KUKA KRL program: MyProgram_286().src

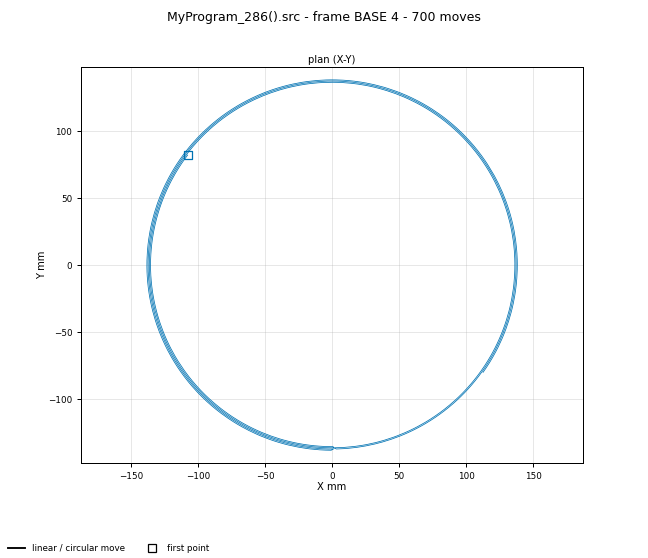
[picture p0: tool path of MyProgram_286().src in frame BASE 4, 700 of 700 moves have a stored position in this frame; points joined in program order, loops and branches not executed]
&ACCESS RVP
&REL 1
&PARAM TEMPLATE = C:\KRC\Roboter\Template\vorgabe
&PARAM EDITMASK = *
DEF MyProgram_286()
; ---- Setting reference (Base) ----
$BASE = BASE_DATA[4]

; --------------------------
; ---- Setting tool (TCP) ----
$TOOL = TOOL_DATA[3]
; --------------------------

$VEL.CP = VEL_APROX_PRINT
Startdeposition()
$VEL.CP = VEL_PRINT
LIN {X -107.8161,Y 82.1036,Z 175,A 144.1909,B 7.7185,C 0.1513,E1 7.5924,E2 307.6378} C_DIS
LIN {X -110.1334,Y 78.9678,Z 175,A 146.0967,B 7.7185,C 0.1516,E1 7.5892,E2 305.7022} C_DIS
LIN {X -112.383,Y 75.7323,Z 175,A 147.6376,B 7.7183,C 0.1573,E1 7.5868,E2 304.1782} C_DIS
LIN {X -114.7272,Y 72.1316,Z 175,A 149.9305,B 7.7183,C 0.1551,E1 7.5833,E2 301.8286} C_DIS
LIN {X -117.0253,Y 68.3406,Z 175,A 151.2224,B 7.7181,C 0.1679,E1 7.5816,E2 300.61} C_DIS
LIN {X -120.0251,Y 62.9181,Z 175,A 153.9854,B 7.718,C 0.1726,E1 7.5779,E2 297.8322} C_DIS
LIN {X -121.646,Y 59.7246,Z 175,A 155.5473,B 7.718,C 0.1759,E1 7.5759,E2 296.2659} C_DIS
LIN {X -123.0692,Y 56.7336,Z 175,A 156.9832,B 7.7179,C 0.179,E1 7.5742,E2 294.8271} C_DIS
LIN {X -124.7084,Y 53.0394,Z 175,A 158.6778,B 7.7177,C 0.1838,E1 7.5723,E2 293.136} C_DIS
LIN {X -126.0542,Y 49.7548,Z 175,A 160.6289,B 7.7177,C 0.1817,E1 7.5703,E2 291.1309} C_DIS
LIN {X -127.3827,Y 46.2436,Z 175,A 162.2434,B 7.7177,C 0.1856,E1 7.5687,E2 289.5146} C_DIS
LIN {X -128.6415,Y 42.6164,Z 175,A 163.4802,B 7.7175,C 0.1953,E1 7.5677,E2 288.327} C_DIS
LIN {X -129.7186,Y 39.2178,Z 175,A 165.0342,B 7.7174,C 0.1989,E1 7.5664,E2 286.7687} C_DIS
LIN {X -130.9414,Y 34.9158,Z 175,A 167.0103,B 7.7173,C 0.203,E1 7.5649,E2 284.7839} C_DIS
LIN {X -131.9367,Y 30.9533,Z 175,A 168.8678,B 7.7172,C 0.2061,E1 7.5637,E2 282.9121} C_DIS
LIN {X -132.7918,Y 27.039,Z 175,A 170.4341,B 7.717,C 0.2126,E1 7.5628,E2 281.363} C_DIS
LIN {X -133.4946,Y 23.33,Z 175,A 172.024,B 7.7169,C 0.2172,E1 7.562,E2 279.7755} C_DIS
LIN {X -134.0907,Y 19.6137,Z 175,A 173.7622,B 7.7169,C 0.2198,E1 7.5613,E2 278.0206} C_DIS
LIN {X -134.5829,Y 15.8836,Z 175,A 175.3324,B 7.7167,C 0.2246,E1 7.5607,E2 276.4544} C_DIS
LIN {X -135.012,Y 11.691,Z 175,A 177.1354,B 7.7165,C 0.2295,E1 7.5602,E2 274.6504} C_DIS
LIN {X -135.2718,Y 8.1499,Z 175,A 178.6452,B 7.7164,C 0.2337,E1 7.56,E2 273.1409} C_DIS
LIN {X -135.4563,Y 4.0677,Z 175,A -179.5523,B 7.7163,C 0.2376,E1 7.5598,E2 271.3307} C_DIS
LIN {X -135.5184,Y 0.2685,Z 175,A -177.968,B 7.7161,C 0.2426,E1 7.5598,E2 269.7506} C_DIS
LIN {X -135.4713,Y -3.5254,Z 175,A -176.2406,B 7.7161,C 0.2455,E1 7.5598,E2 268.0093} C_DIS
LIN {X -135.3015,Y -7.6668,Z 175,A -174.4134,B 7.7159,C 0.2496,E1 7.5601,E2 266.1745} C_DIS
LIN {X -135.0006,Y -11.8252,Z 175,A -172.6182,B 7.7158,C 0.2542,E1 7.5605,E2 264.3766} C_DIS
LIN {X -134.5616,Y -16.0623,Z 175,A -170.8656,B 7.7156,C 0.26,E1 7.561,E2 262.6314} C_DIS
LIN {X -133.9782,Y -20.3659,Z 175,A -168.9506,B 7.7154,C 0.2641,E1 7.5618,E2 260.7082} C_DIS
LIN {X -133.3593,Y -24.0861,Z 175,A -167.4144,B 7.7152,C 0.2694,E1 7.5625,E2 259.1805} C_DIS
LIN {X -132.7048,Y -27.4669,Z 175,A -165.9397,B 7.7152,C 0.2733,E1 7.5633,E2 257.7045} C_DIS
LIN {X -131.904,Y -31.0896,Z 175,A -163.8821,B 7.7152,C 0.2709,E1 7.5647,E2 255.5872} C_DIS
LIN {X -130.9675,Y -34.818,Z 175,A -162.2439,B 7.715,C 0.2752,E1 7.5658,E2 253.9485} C_DIS
LIN {X -129.9083,Y -38.5844,Z 175,A -160.7008,B 7.7148,C 0.2813,E1 7.567,E2 252.4205} C_DIS
LIN {X -128.4088,Y -43.3151,Z 175,A -158.7744,B 7.7145,C 0.2894,E1 7.5687,E2 250.517} C_DIS
LIN {X -127.31,Y -46.4452,Z 175,A -157.4935,B 7.7143,C 0.2948,E1 7.5699,E2 249.2522} C_DIS
LIN {X -126.257,Y -49.2333,Z 175,A -156.1015,B 7.7143,C 0.2963,E1 7.5713,E2 247.8446} C_DIS
LIN {X -124.9108,Y -52.5561,Z 175,A -154.5532,B 7.7141,C 0.2999,E1 7.573,E2 246.2932} C_DIS
LIN {X -123.4445,Y -55.9159,Z 175,A -152.6719,B 7.7141,C 0.2993,E1 7.5752,E2 244.3714} C_DIS
LIN {X -121.9662,Y -59.0717,Z 175,A -151.5247,B 7.7138,C 0.3076,E1 7.5765,E2 243.2659} C_DIS
LIN {X -120.4316,Y -62.1407,Z 175,A -150.0468,B 7.7137,C 0.3109,E1 7.5784,E2 241.7855} C_DIS
LIN {X -117.2772,Y -67.9066,Z 175,A -147.4697,B 7.7133,C 0.3207,E1 7.5818,E2 239.2352} C_DIS
LIN {X -114.8122,Y -71.997,Z 175,A -145.0301,B 7.7133,C 0.3196,E1 7.5854,E2 236.744} C_DIS
LIN {X -110.3112,Y -78.7191,Z 175,A -140.919,B 7.7134,C 0.3176,E1 7.5921,E2 232.5474} C_DIS
LIN {X -106.8941,Y -83.3008,Z 175,A -139.1429,B 7.7128,C 0.3322,E1 7.595,E2 230.8533} C_DIS
LIN {X -104.2988,Y -86.5276,Z 175,A -137.3671,B 7.7127,C 0.3357,E1 7.5981,E2 229.075} C_DIS
LIN {X -101.2925,Y -90.0288,Z 175,A -135.503,B 7.7124,C 0.341,E1 7.6015,E2 227.2226} C_DIS
LIN {X -98.2121,Y -93.3795,Z 175,A -133.4036,B 7.7124,C 0.3424,E1 7.6056,E2 225.1017} C_DIS
LIN {X -95.0625,Y -96.5837,Z 175,A -131.5003,B 7.7122,C 0.3461,E1 7.6093,E2 223.1985} C_DIS
LIN {X -91.4043,Y -100.0534,Z 175,A -129.4346,B 7.712,C 0.3511,E1 7.6135,E2 221.1417} C_DIS
LIN {X -88.3999,Y -102.7166,Z 175,A -127.6314,B 7.712,C 0.3526,E1 7.6173,E2 219.3255} C_DIS
LIN {X -84.3117,Y -106.098,Z 175,A -125.4213,B 7.7117,C 0.357,E1 7.6221,E2 217.1201} C_DIS
LIN {X -81.0086,Y -108.6409,Z 175,A -123.1556,B 7.7119,C 0.3522,E1 7.6273,E2 214.7909} C_DIS
LIN {X -77.435,Y -111.2163,Z 175,A -121.831,B 7.7114,C 0.3634,E1 7.6302,E2 213.5347} C_DIS
LIN {X -74.2923,Y -113.3401,Z 175,A -120.0625,B 7.7114,C 0.3633,E1 7.6343,E2 211.7454} C_DIS
LIN {X -70.4646,Y -115.759,Z 175,A -118.111,B 7.7114,C 0.3654,E1 7.639,E2 209.7894} C_DIS
LIN {X -66.6771,Y -117.981,Z 175,A -116.2393,B 7.7112,C 0.3677,E1 7.6435,E2 207.9158} C_DIS
LIN {X -62.6258,Y -120.1786,Z 175,A -114.4226,B 7.711,C 0.3722,E1 7.648,E2 206.1158} C_DIS
LIN {X -59.8693,Y -121.5745,Z 175,A -113.0442,B 7.711,C 0.3726,E1 7.6514,E2 204.7282} C_DIS
LIN {X -56.0366,Y -123.3904,Z 175,A -111.0915,B 7.711,C 0.372,E1 7.6564,E2 202.7552} C_DIS
LIN {X -52.1981,Y -125.0603,Z 175,A -109.5877,B 7.7107,C 0.3781,E1 7.6602,E2 201.285} C_DIS
LIN {X -48.4755,Y -126.5515,Z 175,A -107.7935,B 7.7107,C 0.3781,E1 7.6649,E2 199.4781} C_DIS
LIN {X -45.5877,Y -127.6192,Z 175,A -106.472,B 7.7107,C 0.3789,E1 7.6684,E2 198.1538} C_DIS
LIN {X -39.2294,Y -129.7151,Z 175,A -103.6522,B 7.7106,C 0.3813,E1 7.6759,E2 195.3351} C_DIS
LIN {X -36.0972,Y -130.6213,Z 175,A -102.2133,B 7.7106,C 0.3813,E1 7.6798,E2 193.8882} C_DIS
LIN {X -32.0637,Y -131.6692,Z 175,A -100.4417,B 7.7106,C 0.3821,E1 7.6846,E2 192.115} C_DIS
LIN {X -28.348,Y -132.5188,Z 175,A -98.8307,B 7.7105,C 0.3829,E1 7.689,E2 190.5035} C_DIS
LIN {X -24.7465,Y -133.24,Z 175,A -97.2309,B 7.7105,C 0.3829,E1 7.6934,E2 188.8974} C_DIS
LIN {X -20.8968,Y -133.896,Z 175,A -95.5882,B 7.7105,C 0.3835,E1 7.6979,E2 187.2552} C_DIS
LIN {X -17.0911,Y -134.4352,Z 175,A -93.628,B 7.7107,C 0.3783,E1 7.7035,E2 185.2516} C_DIS
LIN {X -13.3209,Y -134.8611,Z 175,A -92.3436,B 7.7104,C 0.384,E1 7.7069,E2 184.0075} C_DIS
LIN {X -9.5355,Y -135.1814,Z 175,A -90.5074,B 7.7106,C 0.3803,E1 7.7121,E2 182.1413} C_DIS
LIN {X -6.1557,Y -135.3786,Z 175,A -89.3546,B 7.7104,C 0.385,E1 7.7152,E2 181.0235} C_DIS
LIN {X 0.789,Y -135.5147,Z 175,A -86.4061,B 7.7104,C 0.3846,E1 7.7235,E2 178.0722} C_DIS
LIN {X 0.789,Y -135.5147,Z 175,A -86.4061,B 7.7104,C 0.3846,E1 7.7235,E2 178.0722} C_DIS
Enddeposition()
LIN {X 1.0147,Y -136.4185,Z 175,A -86.3345,B 7.6595,C 0.3899,E1 7.673,E2 178.0513} C_DIS
Startdeposition()
$VEL.CP = VEL_PRINT
LIN {X -5.9801,Y -136.294,Z 175,A -89.7795,B 7.659,C 0.3988,E1 7.6632,E2 181.5627} C_DIS
LIN {X -12.1256,Y -135.885,Z 175,A -92.4451,B 7.659,C 0.3999,E1 7.6557,E2 184.2395} C_DIS
LIN {X -18.4218,Y -135.1756,Z 175,A -95.5048,B 7.6587,C 0.4059,E1 7.6471,E2 187.3506} C_DIS
LIN {X -22.0387,Y -134.632,Z 175,A -96.6557,B 7.659,C 0.399,E1 7.644,E2 188.4533} C_DIS
LIN {X -25.4217,Y -134.0338,Z 175,A -98.1167,B 7.659,C 0.3988,E1 7.64,E2 189.917} C_DIS
LIN {X -28.6784,Y -133.3748,Z 175,A -99.5243,B 7.659,C 0.3983,E1 7.6361,E2 191.3266} C_DIS
LIN {X -31.6236,Y -132.7078,Z 175,A -100.774,B 7.6591,C 0.3973,E1 7.6328,E2 192.5742} C_DIS
LIN {X -34.3363,Y -132.0338,Z 175,A -102.1182,B 7.6591,C 0.3994,E1 7.6291,E2 193.9403} C_DIS
LIN {X -38.6904,Y -130.8222,Z 175,A -103.9583,B 7.6591,C 0.3971,E1 7.6241,E2 195.7734} C_DIS
LIN {X -43.7485,Y -129.2199,Z 175,A -106.2507,B 7.6591,C 0.3964,E1 7.618,E2 198.0744} C_DIS
LIN {X -47.4516,Y -127.9053,Z 175,A -107.7892,B 7.6593,C 0.3932,E1 7.614,E2 199.599} C_DIS
LIN {X -50.3236,Y -126.8042,Z 175,A -109.1767,B 7.6593,C 0.3935,E1 7.6104,E2 200.9987} C_DIS
LIN {X -56.3141,Y -124.2593,Z 175,A -111.941,B 7.6594,C 0.3911,E1 7.6033,E2 203.7671} C_DIS
LIN {X -59.924,Y -122.5584,Z 175,A -113.5022,B 7.6596,C 0.3874,E1 7.5994,E2 205.3139} C_DIS
LIN {X -63.3045,Y -120.846,Z 175,A -115.1161,B 7.6597,C 0.3858,E1 7.5954,E2 206.9306} C_DIS
LIN {X -67.1452,Y -118.7577,Z 175,A -117.04,B 7.6597,C 0.3848,E1 7.5907,E2 208.8656} C_DIS
LIN {X -70.6813,Y -116.6873,Z 175,A -118.7791,B 7.6599,C 0.3827,E1 7.5865,E2 210.607} C_DIS
LIN {X -74.4795,Y -114.3005,Z 175,A -120.7118,B 7.6599,C 0.3807,E1 7.5819,E2 212.5456} C_DIS
LIN {X -78.1156,Y -111.8471,Z 175,A -122.6441,B 7.66,C 0.3792,E1 7.5774,E2 214.489} C_DIS
LIN {X -81.8071,Y -109.1766,Z 175,A -124.5295,B 7.6602,C 0.3757,E1 7.5732,E2 216.3707} C_DIS
LIN {X -85.157,Y -106.5838,Z 175,A -126.196,B 7.6604,C 0.371,E1 7.5696,E2 218.0227} C_DIS
LIN {X -88.185,Y -104.0924,Z 175,A -127.9779,B 7.6604,C 0.3701,E1 7.5657,E2 219.8212} C_DIS
LIN {X -91.4413,Y -101.2439,Z 175,A -129.638,B 7.6607,C 0.3645,E1 7.5623,E2 221.4612} C_DIS
LIN {X -94.0168,Y -98.857,Z 175,A -131.2904,B 7.6607,C 0.3643,E1 7.5589,E2 223.1355} C_DIS
LIN {X -97.1533,Y -95.7764,Z 175,A -133.1996,B 7.6609,C 0.3616,E1 7.5551,E2 225.0521} C_DIS
LIN {X -100.5029,Y -92.2547,Z 175,A -135.1908,B 7.6611,C 0.3567,E1 7.5513,E2 227.0363} C_DIS
LIN {X -103.7292,Y -88.6122,Z 175,A -137.3399,B 7.6612,C 0.3539,E1 7.5473,E2 229.1979} C_DIS
LIN {X -106.6969,Y -85.0149,Z 175,A -139.2989,B 7.6614,C 0.3497,E1 7.5439,E2 231.1562} C_DIS
LIN {X -110.2775,Y -80.3164,Z 175,A -141.8463,B 7.6616,C 0.345,E1 7.5396,E2 233.7109} C_DIS
LIN {X -112.9731,Y -76.4778,Z 175,A -143.9771,B 7.6617,C 0.3427,E1 7.5362,E2 235.8608} C_DIS
LIN {X -115.8349,Y -72.0696,Z 175,A -146.039,B 7.6621,C 0.3354,E1 7.5332,E2 237.9036} C_DIS
LIN {X -118.3923,Y -67.7871,Z 175,A -148.3088,B 7.6621,C 0.3328,E1 7.5299,E2 240.1939} C_DIS
LIN {X -120.522,Y -63.9216,Z 175,A -150.0817,B 7.6624,C 0.327,E1 7.5276,E2 241.9558} C_DIS
LIN {X -122.2542,Y -60.5406,Z 175,A -151.5848,B 7.6626,C 0.3217,E1 7.5257,E2 243.4465} C_DIS
LIN {X -123.5045,Y -57.9521,Z 175,A -152.9385,B 7.6626,C 0.3206,E1 7.5241,E2 244.8177} C_DIS
LIN {X -125.105,Y -54.4064,Z 175,A -154.5088,B 7.6629,C 0.3155,E1 7.5223,E2 246.3792} C_DIS
LIN {X -126.4585,Y -51.1811,Z 175,A -155.9996,B 7.663,C 0.3119,E1 7.5207,E2 247.8716} C_DIS
LIN {X -127.5287,Y -48.4571,Z 175,A -157.1831,B 7.6632,C 0.3081,E1 7.5195,E2 249.0488} C_DIS
LIN {X -128.4332,Y -46.0026,Z 175,A -158.7635,B 7.6631,C 0.3117,E1 7.518,E2 250.688} C_DIS
LIN {X -129.7192,Y -42.2465,Z 175,A -160.0232,B 7.6635,C 0.3016,E1 7.5169,E2 251.8963} C_DIS
LIN {X -132.1456,Y -33.8958,Z 175,A -163.9384,B 7.6637,C 0.2952,E1 7.514,E2 255.8416} C_DIS
LIN {X -133.2218,Y -29.3871,Z 175,A -165.8816,B 7.6639,C 0.2897,E1 7.5127,E2 257.7829} C_DIS
LIN {X -133.9192,Y -26.0215,Z 175,A -167.2777,B 7.6641,C 0.285,E1 7.512,E2 259.172} C_DIS
LIN {X -134.5511,Y -22.5233,Z 175,A -168.7249,B 7.6643,C 0.2802,E1 7.5113,E2 260.6125} C_DIS
LIN {X -135.0574,Y -19.2563,Z 175,A -170.2524,B 7.6643,C 0.2781,E1 7.5106,E2 262.156} C_DIS
LIN {X -135.5764,Y -15.19,Z 175,A -172.0277,B 7.6645,C 0.2739,E1 7.51,E2 263.9366} C_DIS
LIN {X -135.9437,Y -11.4309,Z 175,A -173.5577,B 7.6647,C 0.2686,E1 7.5097,E2 265.4583} C_DIS
LIN {X -136.2347,Y -7.1817,Z 175,A -175.3933,B 7.6648,C 0.2641,E1 7.5093,E2 267.2982} C_DIS
LIN {X -136.3903,Y -3.0903,Z 175,A -177.1761,B 7.665,C 0.26,E1 7.5092,E2 269.0873} C_DIS
LIN {X -136.4227,Y 0.6757,Z 175,A -178.7851,B 7.6651,C 0.2558,E1 7.5092,E2 270.6982} C_DIS
LIN {X -136.3334,Y 4.9675,Z 175,A 179.3984,B 7.6653,C 0.2508,E1 7.5093,E2 272.5148} C_DIS
LIN {X -136.1642,Y 8.4061,Z 175,A 177.8844,B 7.6653,C 0.2475,E1 7.5096,E2 274.0359} C_DIS
LIN {X -135.8582,Y 12.4205,Z 175,A 176.1145,B 7.6655,C 0.2437,E1 7.51,E2 275.8139} C_DIS
LIN {X -135.4751,Y 16.0574,Z 175,A 174.6574,B 7.6657,C 0.2383,E1 7.5104,E2 277.26} C_DIS
LIN {X -135.0275,Y 19.4657,Z 175,A 173.1739,B 7.6657,C 0.2347,E1 7.511,E2 278.7471} C_DIS
LIN {X -134.4643,Y 23.0438,Z 175,A 171.5417,B 7.6659,C 0.2318,E1 7.5117,E2 280.3915} C_DIS
LIN {X -133.7407,Y 26.9221,Z 175,A 169.9244,B 7.666,C 0.2266,E1 7.5126,E2 282.0024} C_DIS
LIN {X -133.097,Y 29.9444,Z 175,A 168.7876,B 7.6662,C 0.2208,E1 7.5133,E2 283.1182} C_DIS
LIN {X -132.3218,Y 33.2017,Z 175,A 167.2123,B 7.6662,C 0.2191,E1 7.5143,E2 284.7129} C_DIS
LIN {X -131.5573,Y 36.1159,Z 175,A 165.9868,B 7.6664,C 0.215,E1 7.5152,E2 285.9324} C_DIS
LIN {X -130.2611,Y 40.5428,Z 175,A 163.9702,B 7.6664,C 0.2107,E1 7.5168,E2 287.9568} C_DIS
LIN {X -126.9378,Y 49.9839,Z 175,A 159.5096,B 7.6667,C 0.2027,E1 7.5211,E2 292.4449} C_DIS
LIN {X -125.4333,Y 53.6471,Z 175,A 158.0078,B 7.6669,C 0.1961,E1 7.5226,E2 293.9254} C_DIS
LIN {X -123.8705,Y 57.1606,Z 175,A 156.3176,B 7.6669,C 0.1928,E1 7.5246,E2 295.6231} C_DIS
LIN {X -122.574,Y 59.8924,Z 175,A 154.9947,B 7.667,C 0.1903,E1 7.5262,E2 296.9513} C_DIS
LIN {X -120.9439,Y 63.1181,Z 175,A 153.4191,B 7.667,C 0.1871,E1 7.5282,E2 298.5324} C_DIS
LIN {X -117.1262,Y 69.9515,Z 175,A 149.9417,B 7.6672,C 0.1814,E1 7.5331,E2 302.0297} C_DIS
LIN {X -114.4716,Y 74.216,Z 175,A 147.8802,B 7.6674,C 0.1756,E1 7.5361,E2 304.0834} C_DIS
LIN {X -111.9926,Y 77.9065,Z 175,A 145.947,B 7.6674,C 0.172,E1 7.5392,E2 306.0227} C_DIS
LIN {X -109.2204,Y 81.7482,Z 175,A 143.9336,B 7.6675,C 0.1677,E1 7.5425,E2 308.0371} C_DIS
LIN {X -106.4146,Y 85.3688,Z 175,A 142.0153,B 7.6676,C 0.1633,E1 7.5458,E2 309.9529} C_DIS
LIN {X -104.1502,Y 88.1169,Z 175,A 140.3864,B 7.6676,C 0.1618,E1 7.5488,E2 311.5966} C_DIS
LIN {X -100.7665,Y 91.9675,Z 175,A 138.2088,B 7.6678,C 0.1575,E1 7.5528,E2 313.7751} C_DIS
LIN {X -97.3769,Y 95.5484,Z 175,A 136.2701,B 7.6678,C 0.1513,E1 7.5566,E2 315.6959} C_DIS
LIN {X -95.1526,Y 97.7644,Z 175,A 134.834,B 7.6678,C 0.1503,E1 7.5594,E2 317.1449} C_DIS
LIN {X -91.7325,Y 100.9798,Z 175,A 133.0706,B 7.668,C 0.1435,E1 7.563,E2 318.8814} C_DIS
LIN {X -88.465,Y 103.8543,Z 175,A 131.0391,B 7.668,C 0.1429,E1 7.5673,E2 320.9359} C_DIS
LIN {X -84.5576,Y 107.0603,Z 175,A 128.7776,B 7.668,C 0.141,E1 7.5723,E2 323.2123} C_DIS
LIN {X -81.7923,Y 109.1876,Z 175,A 126.7669,B 7.668,C 0.1462,E1 7.577,E2 325.2871} C_DIS
LIN {X -77.3033,Y 112.4099,Z 175,A 125.0892,B 7.6682,C 0.1332,E1 7.5806,E2 326.8857} C_DIS
LIN {X -73.7646,Y 114.7633,Z 175,A 123.2589,B 7.6682,C 0.131,E1 7.5849,E2 328.72} C_DIS
LIN {X -70.1868,Y 116.986,Z 175,A 121.0945,B 7.6682,C 0.1341,E1 7.5902,E2 330.9306} C_DIS
LIN {X -66.6098,Y 119.0587,Z 175,A 119.7164,B 7.6683,C 0.1264,E1 7.5934,E2 332.2642} C_DIS
LIN {X -62.6935,Y 121.1669,Z 175,A 117.9297,B 7.6683,C 0.1227,E1 7.5978,E2 334.0395} C_DIS
LIN {X -58.2166,Y 123.3794,Z 175,A 115.7073,B 7.6683,C 0.1219,E1 7.6034,E2 336.2754} C_DIS
LIN {X -54.468,Y 125.0783,Z 175,A 114.0896,B 7.6685,C 0.1182,E1 7.6075,E2 337.8784} C_DIS
LIN {X -51.7249,Y 126.2393,Z 175,A 112.8302,B 7.6685,C 0.1169,E1 7.6107,E2 339.138} C_DIS
LIN {X -48.0338,Y 127.6872,Z 175,A 111.2793,B 7.6685,C 0.1134,E1 7.6147,E2 340.6737} C_DIS
LIN {X -45.6207,Y 128.5709,Z 175,A 109.8649,B 7.6685,C 0.1175,E1 7.6186,E2 342.1279} C_DIS
LIN {X -41.9386,Y 129.8176,Z 175,A 108.3515,B 7.6685,C 0.1142,E1 7.6225,E2 343.6257} C_DIS
LIN {X -39.0384,Y 130.7203,Z 175,A 106.9717,B 7.6685,C 0.1147,E1 7.6263,E2 345.0173} C_DIS
LIN {X -34.3874,Y 132.0204,Z 175,A 104.9365,B 7.6685,C 0.1133,E1 7.6317,E2 347.052} C_DIS
LIN {X -30.7554,Y 132.9118,Z 175,A 103.5377,B 7.6685,C 0.1096,E1 7.6355,E2 348.429} C_DIS
LIN {X -27.2768,Y 133.6685,Z 175,A 101.9915,B 7.6685,C 0.1095,E1 7.6397,E2 349.9804} C_DIS
LIN {X -24.2915,Y 134.2434,Z 175,A 100.8185,B 7.6686,C 0.1071,E1 7.6429,E2 351.1401} C_DIS
LIN {X -21.0093,Y 134.7959,Z 175,A 99.2883,B 7.6686,C 0.1086,E1 7.6472,E2 352.6856} C_DIS
LIN {X -17.4113,Y 135.3081,Z 175,A 97.7067,B 7.6686,C 0.1089,E1 7.6516,E2 354.273} C_DIS
LIN {X -13.673,Y 135.738,Z 175,A 96.1105,B 7.6686,C 0.1086,E1 7.656,E2 355.8703} C_DIS
LIN {X -10.5237,Y 136.0182,Z 175,A 94.7698,B 7.6686,C 0.1086,E1 7.6597,E2 357.2118} C_DIS
LIN {X -6.7796,Y 136.2549,Z 175,A 93.243,B 7.6686,C 0.1075,E1 7.664,E2 358.7319} C_DIS
LIN {X -2.5961,Y 136.3992,Z 175,A 91.7279,B 7.6686,C 0.1034,E1 7.6681,E2 360.2168} C_DIS
LIN {X 0.4564,Y 136.4231,Z 175,A 89.9308,B 7.6686,C 0.1117,E1 7.6733,E2 362.0755} C_DIS
LIN {X 3.8305,Y 136.3697,Z 175,A 88.4641,B 7.6686,C 0.1126,E1 7.6774,E2 363.5476} C_DIS
LIN {X 7.6414,Y 136.2113,Z 175,A 87.1087,B 7.6686,C 0.1089,E1 7.6811,E2 364.8727} C_DIS
LIN {X 11.4052,Y 135.9458,Z 175,A 85.8168,B 7.6686,C 0.1044,E1 7.6846,E2 366.1285} C_DIS
LIN {X 14.6117,Y 135.6386,Z 175,A 84.2516,B 7.6686,C 0.1083,E1 7.689,E2 367.7189} C_DIS
LIN {X 19.2039,Y 135.0649,Z 175,A 82.3801,B 7.6686,C 0.1078,E1 7.6942,E2 369.5811} C_DIS
LIN {X 22.3419,Y 134.5814,Z 175,A 81.025,B 7.6686,C 0.1088,E1 7.6979,E2 370.9384} C_DIS
LIN {X 25.7005,Y 133.9805,Z 175,A 79.6424,B 7.6686,C 0.1087,E1 7.7017,E2 372.3144} C_DIS
LIN {X 28.2187,Y 133.4741,Z 175,A 78.505,B 7.6686,C 0.1103,E1 7.7048,E2 373.4588} C_DIS
LIN {X 31.8089,Y 132.6631,Z 175,A 76.9798,B 7.6686,C 0.1109,E1 7.709,E2 374.9811} C_DIS
LIN {X 35.3746,Y 131.7572,Z 175,A 75.388,B 7.6686,C 0.1129,E1 7.7133,E2 376.5782} C_DIS
LIN {X 40.758,Y 130.1947,Z 175,A 72.9885,B 7.6685,C 0.1156,E1 7.7197,E2 378.9828} C_DIS
LIN {X 44.4703,Y 128.9716,Z 175,A 71.4569,B 7.6685,C 0.1152,E1 7.7237,E2 380.5007} C_DIS
LIN {X 47.376,Y 127.9336,Z 175,A 70.0763,B 7.6685,C 0.1179,E1 7.7274,E2 381.8915} C_DIS
LIN {X 53.2389,Y 125.608,Z 175,A 67.4297,B 7.6685,C 0.1207,E1 7.7342,E2 384.5375} C_DIS
LIN {X 56.8976,Y 123.9921,Z 175,A 65.8616,B 7.6685,C 0.1207,E1 7.7382,E2 386.0919} C_DIS
LIN {X 60.4223,Y 122.3126,Z 175,A 64.2892,B 7.6684,C 0.1216,E1 7.7421,E2 387.6561} C_DIS
LIN {X 62.8063,Y 121.1076,Z 175,A 63.0725,B 7.6684,C 0.1248,E1 7.7452,E2 388.8844} C_DIS
LIN {X 66.603,Y 119.0625,Z 175,A 61.2749,B 7.6684,C 0.127,E1 7.7496,E2 390.6804} C_DIS
LIN {X 70.3552,Y 116.8845,Z 175,A 59.4473,B 7.6683,C 0.1298,E1 7.754,E2 392.5088} C_DIS
LIN {X 74.0665,Y 114.5687,Z 175,A 57.6112,B 7.6683,C 0.1326,E1 7.7583,E2 394.3448} C_DIS
LIN {X 77.7122,Y 112.1278,Z 175,A 55.7938,B 7.6682,C 0.1351,E1 7.7625,E2 396.1593} C_DIS
LIN {X 81.3742,Y 109.4989,Z 175,A 53.9506,B 7.6682,C 0.1374,E1 7.7666,E2 397.9968} C_DIS
LIN {X 84.9439,Y 106.7534,Z 175,A 52.0943,B 7.6681,C 0.1401,E1 7.7707,E2 399.8491} C_DIS
LIN {X 88.3954,Y 103.9135,Z 175,A 50.2509,B 7.6681,C 0.1429,E1 7.7746,E2 401.6888} C_DIS
LIN {X 91.6243,Y 101.0779,Z 175,A 48.4627,B 7.668,C 0.146,E1 7.7784,E2 403.4753} C_DIS
LIN {X 94.7513,Y 98.1529,Z 175,A 46.6628,B 7.668,C 0.1496,E1 7.782,E2 405.2759} C_DIS
LIN {X 97.9117,Y 95.0005,Z 175,A 44.8119,B 7.6678,C 0.153,E1 7.7856,E2 407.1245} C_DIS
LIN {X 101.0729,Y 91.6298,Z 175,A 42.9202,B 7.6678,C 0.1561,E1 7.7892,E2 409.0108} C_DIS
LIN {X 104.0652,Y 88.2169,Z 175,A 41.0489,B 7.6678,C 0.1596,E1 7.7926,E2 410.8785} C_DIS
LIN {X 107.1202,Y 84.4813,Z 175,A 39.0236,B 7.6676,C 0.1641,E1 7.7962,E2 412.9044} C_DIS
LIN {X 109.7989,Y 80.9692,Z 175,A 37.1752,B 7.6676,C 0.1682,E1 7.7993,E2 414.7527} C_DIS
LIN {X 112.3569,Y 77.3804,Z 175,A 35.3546,B 7.6674,C 0.172,E1 7.8022,E2 416.5705} C_DIS
LIN {X 114.9549,Y 73.4653,Z 175,A 33.4428,B 7.6674,C 0.1756,E1 7.8051,E2 418.4756} C_DIS
LIN {X 117.3056,Y 69.6507,Z 175,A 31.5851,B 7.6673,C 0.1797,E1 7.8078,E2 420.3313} C_DIS
LIN {X 119.4892,Y 65.8344,Z 175,A 29.7643,B 7.6672,C 0.1838,E1 7.8103,E2 422.1499} C_DIS
LIN {X 121.425,Y 62.1876,Z 175,A 28.1238,B 7.6672,C 0.1864,E1 7.8124,E2 423.7797} C_DIS
LIN {X 122.987,Y 59.0379,Z 175,A 26.7622,B 7.6671,C 0.188,E1 7.814,E2 425.128} C_DIS
LIN {X 124.3459,Y 56.1205,Z 175,A 25.3614,B 7.667,C 0.1925,E1 7.8157,E2 426.5357} C_DIS
LIN {X 125.7124,Y 52.9888,Z 175,A 23.8484,B 7.6668,C 0.1978,E1 7.8173,E2 428.0592} C_DIS
LIN {X 127.0288,Y 49.7496,Z 175,A 22.119,B 7.6666,C 0.2067,E1 7.8192,E2 429.8217} C_DIS
LIN {X 128.3892,Y 46.1247,Z 175,A 20.8852,B 7.6666,C 0.2035,E1 7.8203,E2 431.0082} C_DIS
LIN {X 129.7484,Y 42.1552,Z 175,A 19.1156,B 7.6666,C 0.2085,E1 7.8218,E2 432.78} C_DIS
LIN {X 130.8233,Y 38.6865,Z 175,A 17.6624,B 7.6665,C 0.2113,E1 7.823,E2 434.2253} C_DIS
LIN {X 131.7291,Y 35.4801,Z 175,A 16.2706,B 7.6664,C 0.215,E1 7.824,E2 435.6172} C_DIS
LIN {X 132.5574,Y 32.2473,Z 175,A 15.0548,B 7.6664,C 0.2152,E1 7.8249,E2 436.8109} C_DIS
LIN {X 133.1955,Y 29.5093,Z 175,A 13.6097,B 7.6661,C 0.2237,E1 7.8258,E2 438.2898} C_DIS
LIN {X 134.0628,Y 25.2702,Z 175,A 11.9013,B 7.6661,C 0.2267,E1 7.8267,E2 439.986} C_DIS
LIN {X 134.7769,Y 21.1324,Z 175,A 10.3263,B 7.666,C 0.228,E1 7.8274,E2 441.539} C_DIS
LIN {X 135.1757,Y 18.4211,Z 175,A 9.0192,B 7.6658,C 0.2344,E1 7.8279,E2 442.8664} C_DIS
LIN {X 135.6387,Y 14.6112,Z 175,A 7.5661,B 7.6658,C 0.2359,E1 7.8284,E2 444.301} C_DIS
LIN {X 135.9755,Y 11.0542,Z 175,A 5.9609,B 7.6656,C 0.2422,E1 7.8287,E2 445.9205} C_DIS
LIN {X 136.3311,Y 5.0287,Z 175,A 3.5933,B 7.6654,C 0.2462,E1 7.8291,E2 448.2695} C_DIS
LIN {X 136.418,Y 1.3992,Z 175,A 1.9358,B 7.6652,C 0.2532,E1 7.8291,E2 449.9448} C_DIS
LIN {X 136.3923,Y -3.011,Z 175,A 0.3186,B 7.6652,C 0.2539,E1 7.8291,E2 451.5343} C_DIS
LIN {X 136.23,Y -7.2749,Z 175,A -1.5647,B 7.6649,C 0.2609,E1 7.8289,E2 453.4306} C_DIS
LIN {X 135.723,Y -13.8275,Z 175,A -4.3207,B 7.6647,C 0.2688,E1 7.8282,E2 456.1886} C_DIS
LIN {X 135.2708,Y -17.6953,Z 175,A -5.8241,B 7.6647,C 0.2708,E1 7.8277,E2 457.6769} C_DIS
LIN {X 134.6441,Y -21.9664,Z 175,A -7.5752,B 7.6645,C 0.2748,E1 7.827,E2 459.4219} C_DIS
LIN {X 134.1621,Y -24.7457,Z 175,A -8.8739,B 7.6643,C 0.2805,E1 7.8263,E2 460.7361} C_DIS
LIN {X 133.3414,Y -28.8333,Z 175,A -10.3423,B 7.6643,C 0.2798,E1 7.8255,E2 462.1707} C_DIS
LIN {X 132.7818,Y -31.3164,Z 175,A -11.4298,B 7.6642,C 0.2832,E1 7.8248,E2 463.2616} C_DIS
LIN {X 131.9438,Y -34.6747,Z 175,A -12.7917,B 7.6641,C 0.2855,E1 7.8239,E2 464.6133} C_DIS
LIN {X 131.0023,Y -38.0755,Z 175,A -14.3643,B 7.6639,C 0.2914,E1 7.8227,E2 466.1988} C_DIS
LIN {X 130.1414,Y -40.9249,Z 175,A -15.5197,B 7.6638,C 0.293,E1 7.8217,E2 467.3435} C_DIS
LIN {X 129.0005,Y -44.387,Z 175,A -17.0575,B 7.6636,C 0.2974,E1 7.8204,E2 468.8836} C_DIS
LIN {X 127.8481,Y -47.6043,Z 175,A -18.554,B 7.6634,C 0.3025,E1 7.8189,E2 470.3892} C_DIS
LIN {X 126.5061,Y -51.063,Z 175,A -20.0455,B 7.6634,C 0.3054,E1 7.8174,E2 471.8738} C_DIS
LIN {X 125.0056,Y -54.6362,Z 175,A -21.883,B 7.663,C 0.3139,E1 7.8154,E2 473.7394} C_DIS
LIN {X 123.342,Y -58.2948,Z 175,A -23.2034,B 7.663,C 0.3112,E1 7.8139,E2 475.0152} C_DIS
LIN {X 121.6896,Y -61.6678,Z 175,A -24.9168,B 7.6628,C 0.318,E1 7.8117,E2 476.7472} C_DIS
LIN {X 119.9014,Y -65.0807,Z 175,A -26.5109,B 7.6626,C 0.3217,E1 7.8096,E2 478.3401} C_DIS
LIN {X 118.172,Y -68.1702,Z 175,A -28.0118,B 7.6625,C 0.3258,E1 7.8075,E2 479.8441} C_DIS
LIN {X 116.3404,Y -71.2509,Z 175,A -29.852,B 7.662,C 0.3361,E1 7.8048,E2 481.7279} C_DIS
LIN {X 114.0753,Y -74.8241,Z 175,A -31.2477,B 7.6622,C 0.3331,E1 7.8027,E2 483.0775} C_DIS
LIN {X 111.2186,Y -79.0086,Z 175,A -33.285,B 7.662,C 0.3365,E1 7.7995,E2 485.1055} C_DIS
LIN {X 108.6719,Y -82.4762,Z 175,A -35.0656,B 7.6619,C 0.3403,E1 7.7965,E2 486.8846} C_DIS
LIN {X 106.0108,Y -85.8694,Z 175,A -36.7201,B 7.6618,C 0.3414,E1 7.7937,E2 488.5211} C_DIS
LIN {X 103.7234,Y -88.619,Z 175,A -38.3802,B 7.6615,C 0.3479,E1 7.7907,E2 490.2026} C_DIS
LIN {X 100.7821,Y -91.9504,Z 175,A -40.2021,B 7.6614,C 0.3512,E1 7.7873,E2 492.0206} C_DIS
LIN {X 97.7144,Y -95.2042,Z 175,A -42.0811,B 7.6612,C 0.3552,E1 7.7837,E2 493.9015} C_DIS
LIN {X 94.5454,Y -98.3518,Z 175,A -43.9112,B 7.661,C 0.3583,E1 7.78,E2 495.7276} C_DIS
LIN {X 91.9401,Y -100.7914,Z 175,A -45.4431,B 7.6609,C 0.3619,E1 7.7769,E2 497.2651} C_DIS
LIN {X 87.8155,Y -104.4041,Z 175,A -47.6771,B 7.6607,C 0.3651,E1 7.7721,E2 499.4925} C_DIS
LIN {X 84.1045,Y -107.4162,Z 175,A -49.5855,B 7.6607,C 0.3671,E1 7.768,E2 501.3902} C_DIS
LIN {X 80.6452,Y -110.037,Z 175,A -51.4431,B 7.6604,C 0.371,E1 7.7638,E2 503.2539} C_DIS
LIN {X 77.0714,Y -112.569,Z 175,A -53.2648,B 7.6603,C 0.3739,E1 7.7597,E2 505.075} C_DIS
LIN {X 73.2654,Y -115.0828,Z 175,A -55.0766,B 7.6603,C 0.3751,E1 7.7554,E2 506.8753} C_DIS
LIN {X 69.4198,Y -117.4426,Z 175,A -57.7704,B 7.6593,C 0.3929,E1 7.7487,E2 509.6714} C_DIS
LIN {X 64.0371,Y -120.4613,Z 175,A -59.4481,B 7.66,C 0.3799,E1 7.7449,E2 511.236} C_DIS
LIN {X 61.3402,Y -121.8563,Z 175,A -60.9369,B 7.6597,C 0.3856,E1 7.7411,E2 512.7529} C_DIS
LIN {X 58.0392,Y -123.4628,Z 175,A -62.3289,B 7.6597,C 0.385,E1 7.7376,E2 514.1272} C_DIS
LIN {X 54.446,Y -125.0878,Z 175,A -63.9509,B 7.6597,C 0.3864,E1 7.7335,E2 515.7461} C_DIS
LIN {X 51.2115,Y -126.4463,Z 175,A -65.4194,B 7.6596,C 0.3881,E1 7.7297,E2 517.2151} C_DIS
LIN {X 48.5142,Y -127.5073,Z 175,A -66.5569,B 7.6596,C 0.3881,E1 7.7268,E2 518.3435} C_DIS
LIN {X 45.6796,Y -128.5496,Z 175,A -67.9895,B 7.6594,C 0.3924,E1 7.723,E2 519.7979} C_DIS
LIN {X 41.9537,Y -129.8127,Z 175,A -69.4562,B 7.6594,C 0.3908,E1 7.7191,E2 521.2421} C_DIS
LIN {X 39.193,Y -130.6742,Z 175,A -70.8519,B 7.6592,C 0.3952,E1 7.7153,E2 522.6618} C_DIS
LIN {X 35.474,Y -131.7307,Z 175,A -72.362,B 7.6592,C 0.3946,E1 7.7113,E2 524.1585} C_DIS
LIN {X 32.0915,Y -132.595,Z 175,A -73.7997,B 7.6592,C 0.3953,E1 7.7074,E2 525.5936} C_DIS
LIN {X 28.8435,Y -133.3392,Z 175,A -75.0391,B 7.6593,C 0.3935,E1 7.7041,E2 526.8135} C_DIS
LIN {X 26.2553,Y -133.8745,Z 175,A -76.4054,B 7.659,C 0.3988,E1 7.7003,E2 528.2132} C_DIS
LIN {X 22.5866,Y -134.5406,Z 175,A -77.8032,B 7.6591,C 0.3968,E1 7.6965,E2 529.5904} C_DIS
LIN {X 16.8218,Y -135.3839,Z 175,A -80.2174,B 7.6591,C 0.3975,E1 7.6898,E2 532.0021} C_DIS
LIN {X 8.4085,Y -136.1641,Z 175,A -83.8584,B 7.659,C 0.4004,E1 7.6797,E2 535.6568} C_DIS
LIN {X 1.0147,Y -136.4185,Z 175,A -85.6162,B 7.6601,C 0.3779,E1 7.6753,E2 537.2433} C_DIS
Enddeposition()
LIN {X 1.0147,Y -136.4185,Z 175,A -85.6165,B 7.6601,C 0.3779,E1 7.6753,E2 537.2436} C_DIS
Startdeposition()
$VEL.CP = VEL_PRINT
LIN {X 3.26,Y -137.2924,Z 175,A -85.4246,B 7.6096,C 0.3955,E1 7.6258,E2 537.1951} C_DIS
LIN {X 6.3358,Y -137.1849,Z 175,A -83.9811,B 7.6098,C 0.3924,E1 7.6299,E2 535.7304} C_DIS
LIN {X 9.2202,Y -137.0223,Z 175,A -82.7861,B 7.6098,C 0.3922,E1 7.6332,E2 534.5361} C_DIS
LIN {X 12.3399,Y -136.7766,Z 175,A -81.5519,B 7.6098,C 0.393,E1 7.6366,E2 533.3104} C_DIS
LIN {X 15.8307,Y -136.415,Z 175,A -80.2197,B 7.6097,C 0.3946,E1 7.6403,E2 531.9944} C_DIS
LIN {X 18.6353,Y -136.0619,Z 175,A -78.8395,B 7.6099,C 0.3905,E1 7.6442,E2 530.5876} C_DIS
LIN {X 22.0259,Y -135.5532,Z 175,A -77.4837,B 7.6099,C 0.391,E1 7.6479,E2 529.2406} C_DIS
LIN {X 24.9894,Y -135.0394,Z 175,A -76.1597,B 7.6099,C 0.389,E1 7.6516,E2 527.9069} C_DIS
LIN {X 28.759,Y -134.2848,Z 175,A -74.6251,B 7.6099,C 0.3891,E1 7.6557,E2 526.3802} C_DIS
LIN {X 31.8454,Y -133.5867,Z 175,A -73.3948,B 7.6099,C 0.3897,E1 7.6591,E2 525.1607} C_DIS
LIN {X 34.5841,Y -132.9062,Z 175,A -72.1453,B 7.61,C 0.3875,E1 7.6625,E2 523.9011} C_DIS
LIN {X 37.7881,Y -132.031,Z 175,A -70.6908,B 7.6102,C 0.385,E1 7.6664,E2 522.4368} C_DIS
LIN {X 41.2107,Y -131.0017,Z 175,A -69.2819,B 7.6102,C 0.385,E1 7.6701,E2 521.0374} C_DIS
LIN {X 44.1864,Y -130.0295,Z 175,A -67.9832,B 7.6102,C 0.3838,E1 7.6736,E2 519.7388} C_DIS
LIN {X 47.5942,Y -128.8199,Z 175,A -66.4833,B 7.6102,C 0.3823,E1 7.6775,E2 518.2388} C_DIS
LIN {X 50.5512,Y -127.6898,Z 175,A -65.0445,B 7.6105,C 0.3786,E1 7.6813,E2 516.7837} C_DIS
LIN {X 53.7477,Y -126.3773,Z 175,A -63.6757,B 7.6105,C 0.3782,E1 7.6848,E2 515.4233} C_DIS
LIN {X 56.8566,Y -125.0098,Z 175,A -62.3335,B 7.6105,C 0.3778,E1 7.6882,E2 514.0896} C_DIS
LIN {X 59.9786,Y -123.5422,Z 175,A -60.8285,B 7.6107,C 0.3746,E1 7.692,E2 512.575} C_DIS
LIN {X 63.3133,Y -121.8653,Z 175,A -59.4236,B 7.6107,C 0.3753,E1 7.6955,E2 511.1886} C_DIS
LIN {X 66.8021,Y -119.9896,Z 175,A -57.6796,B 7.6108,C 0.3711,E1 7.6998,E2 509.4313} C_DIS
LIN {X 70.0403,Y -118.1286,Z 175,A -56.1802,B 7.6109,C 0.3698,E1 7.7034,E2 507.9383} C_DIS
LIN {X 73.5697,Y -115.9634,Z 175,A -54.4258,B 7.6111,C 0.3665,E1 7.7076,E2 506.1789} C_DIS
LIN {X 77.2227,Y -113.5634,Z 175,A -52.6491,B 7.6111,C 0.3643,E1 7.7117,E2 504.4066} C_DIS
LIN {X 80.3342,Y -111.3842,Z 175,A -51.0986,B 7.6113,C 0.3622,E1 7.7152,E2 502.8592} C_DIS
LIN {X 83.6838,Y -108.89,Z 175,A -49.3632,B 7.6114,C 0.3591,E1 7.7191,E2 501.1231} C_DIS
LIN {X 87.001,Y -106.258,Z 175,A -47.5582,B 7.6116,C 0.355,E1 7.723,E2 499.3116} C_DIS
LIN {X 90.5345,Y -103.2643,Z 175,A -45.679,B 7.6117,C 0.3523,E1 7.727,E2 497.4373} C_DIS
LIN {X 93.3555,Y -100.7212,Z 175,A -44.1599,B 7.6118,C 0.3503,E1 7.7301,E2 495.9253} C_DIS
LIN {X 95.931,Y -98.2713,Z 175,A -42.5798,B 7.6121,C 0.3454,E1 7.7333,E2 494.3312} C_DIS
LIN {X 98.9755,Y -95.2049,Z 175,A -40.9195,B 7.6121,C 0.3443,E1 7.7365,E2 492.6876} C_DIS
LIN {X 101.4061,Y -92.6117,Z 175,A -39.4269,B 7.6123,C 0.3409,E1 7.7393,E2 491.1923} C_DIS
LIN {X 104.2666,Y -89.3783,Z 175,A -37.6071,B 7.6125,C 0.3365,E1 7.7427,E2 489.3684} C_DIS
LIN {X 107.0978,Y -85.9656,Z 175,A -35.8489,B 7.6125,C 0.334,E1 7.7458,E2 487.6203} C_DIS
LIN {X 109.427,Y -82.9805,Z 175,A -34.1912,B 7.6128,C 0.3288,E1 7.7486,E2 485.9509} C_DIS
LIN {X 112.0395,Y -79.4177,Z 175,A -32.4939,B 7.6128,C 0.3272,E1 7.7513,E2 484.2706} C_DIS
LIN {X 114.3951,Y -75.9853,Z 175,A -30.7416,B 7.613,C 0.3227,E1 7.7541,E2 482.5147} C_DIS
LIN {X 116.4313,Y -72.827,Z 175,A -29.2445,B 7.6131,C 0.3202,E1 7.7563,E2 481.0251} C_DIS
LIN {X 118.5723,Y -69.2866,Z 175,A -27.5351,B 7.6133,C 0.3162,E1 7.7588,E2 479.3161} C_DIS
LIN {X 120.3535,Y -66.145,Z 175,A -25.9491,B 7.6135,C 0.3107,E1 7.7609,E2 477.7185} C_DIS
LIN {X 121.9899,Y -63.0759,Z 175,A -24.5665,B 7.6136,C 0.3083,E1 7.7627,E2 476.3433} C_DIS
LIN {X 123.645,Y -59.7635,Z 175,A -23.126,B 7.6137,C 0.3063,E1 7.7645,E2 474.9146} C_DIS
LIN {X 125.0098,Y -56.8566,Z 175,A -21.7351,B 7.6139,C 0.3018,E1 7.7661,E2 473.5159} C_DIS
LIN {X 126.4834,Y -53.4949,Z 175,A -20.2558,B 7.614,C 0.2987,E1 7.7677,E2 472.0418} C_DIS
LIN {X 127.7206,Y -50.4719,Z 175,A -19.0015,B 7.614,C 0.2972,E1 7.769,E2 470.8} C_DIS
LIN {X 128.9814,Y -47.1547,Z 175,A -17.5188,B 7.6142,C 0.2931,E1 7.7705,E2 469.3156} C_DIS
LIN {X 130.0295,Y -44.1864,Z 175,A -16.2302,B 7.6144,C 0.29,E1 7.7716,E2 468.0289} C_DIS
LIN {X 131.0723,Y -40.9899,Z 175,A -14.7814,B 7.6145,C 0.2851,E1 7.7729,E2 466.5729} C_DIS
LIN {X 132.0928,Y -37.5668,Z 175,A -13.3941,B 7.6146,C 0.283,E1 7.7739,E2 465.1973} C_DIS
LIN {X 132.9913,Y -34.2486,Z 175,A -12.1132,B 7.6146,C 0.2821,E1 7.7748,E2 463.9346} C_DIS
LIN {X 133.6987,Y -31.3811,Z 175,A -10.7071,B 7.6149,C 0.2751,E1 7.7758,E2 462.5052} C_DIS
LIN {X 134.5255,Y -27.6115,Z 175,A -9.3095,B 7.6149,C 0.2748,E1 7.7766,E2 461.1331} C_DIS
LIN {X 135.0394,Y -24.9894,Z 175,A -8.1103,B 7.6151,C 0.27,E1 7.7772,E2 459.9222} C_DIS
LIN {X 135.5898,Y -21.8063,Z 175,A -6.7197,B 7.6152,C 0.2652,E1 7.7778,E2 458.5249} C_DIS
LIN {X 136.0905,Y -18.4171,Z 175,A -5.2936,B 7.6154,C 0.2612,E1 7.7784,E2 457.0978} C_DIS
LIN {X 136.4804,Y -15.262,Z 175,A -4.091,B 7.6154,C 0.2599,E1 7.7788,E2 455.9098} C_DIS
LIN {X 136.7766,Y -12.3399,Z 175,A -2.8224,B 7.6156,C 0.2555,E1 7.7791,E2 454.6346} C_DIS
LIN {X 137.0355,Y -9.0059,Z 175,A -1.4473,B 7.6156,C 0.2519,E1 7.7794,E2 453.2608} C_DIS
LIN {X 137.2039,Y -5.9096,Z 175,A -0.3345,B 7.6157,C 0.2518,E1 7.7795,E2 452.1699} C_DIS
LIN {X 137.2983,Y -3.0482,Z 175,A 1.057,B 7.6159,C 0.2444,E1 7.7796,E2 450.7523} C_DIS
LIN {X 137.3282,Y 0.8688,Z 175,A 2.6068,B 7.616,C 0.2414,E1 7.7796,E2 449.2117} C_DIS
LIN {X 137.2557,Y 4.5821,Z 175,A 4.1992,B 7.6162,C 0.236,E1 7.7796,E2 447.6126} C_DIS
LIN {X 137.0223,Y 9.2202,Z 175,A 6.012,B 7.6162,C 0.233,E1 7.7792,E2 445.814} C_DIS
LIN {X 136.7766,Y 12.3399,Z 175,A 7.226,B 7.6164,C 0.231,E1 7.7789,E2 444.6107} C_DIS
LIN {X 136.457,Y 15.4791,Z 175,A 8.5205,B 7.6164,C 0.2277,E1 7.7785,E2 443.3179} C_DIS
LIN {X 136.0619,Y 18.6353,Z 175,A 9.8959,B 7.6166,C 0.223,E1 7.778,E2 441.9353} C_DIS
LIN {X 135.5532,Y 22.0259,Z 175,A 11.2818,B 7.6166,C 0.2198,E1 7.7774,E2 440.5539} C_DIS
LIN {X 134.9469,Y 25.4734,Z 175,A 12.5855,B 7.6167,C 0.2188,E1 7.7768,E2 439.2689} C_DIS
LIN {X 134.4094,Y 28.1819,Z 175,A 13.8717,B 7.6169,C 0.2129,E1 7.7761,E2 437.9648} C_DIS
LIN {X 133.6454,Y 31.6022,Z 175,A 15.237,B 7.6169,C 0.2107,E1 7.7752,E2 436.6107} C_DIS
LIN {X 132.8514,Y 34.7896,Z 175,A 16.6097,B 7.617,C 0.2068,E1 7.7743,E2 435.2368} C_DIS
LIN {X 131.9197,Y 38.1682,Z 175,A 17.9715,B 7.6171,C 0.2048,E1 7.7732,E2 433.8865} C_DIS
LIN {X 131.0017,Y 41.2107,Z 175,A 19.3903,B 7.6172,C 0.1993,E1 7.772,E2 432.4552} C_DIS
LIN {X 129.9079,Y 44.5372,Z 175,A 20.7334,B 7.6172,C 0.1977,E1 7.7709,E2 431.1259} C_DIS
LIN {X 128.8199,Y 47.5942,Z 175,A 22.0943,B 7.6174,C 0.1939,E1 7.7696,E2 429.7632} C_DIS
LIN {X 127.5913,Y 50.7957,Z 175,A 23.4053,B 7.6174,C 0.1924,E1 7.7682,E2 428.4665} C_DIS
LIN {X 126.3924,Y 53.713,Z 175,A 24.8718,B 7.6176,C 0.186,E1 7.7666,E2 426.9802} C_DIS
LIN {X 124.9298,Y 57.0295,Z 175,A 26.3742,B 7.6176,C 0.1822,E1 7.7649,E2 425.4781} C_DIS
LIN {X 123.5422,Y 59.9786,Z 175,A 27.6983,B 7.6177,C 0.1794,E1 7.7633,E2 424.1578} C_DIS
LIN {X 121.8784,Y 63.2883,Z 175,A 29.2034,B 7.6178,C 0.1763,E1 7.7614,E2 422.6568} C_DIS
LIN {X 119.8722,Y 67.0124,Z 175,A 30.8797,B 7.6178,C 0.1735,E1 7.7592,E2 420.9907} C_DIS
LIN {X 118.1286,Y 70.0403,Z 175,A 32.3148,B 7.6179,C 0.1704,E1 7.7572,E2 419.5577} C_DIS
LIN {X 115.9634,Y 73.5697,Z 175,A 34.088,B 7.6181,C 0.1653,E1 7.7545,E2 417.7779} C_DIS
LIN {X 113.9057,Y 76.7171,Z 175,A 35.6771,B 7.6181,C 0.1612,E1 7.7521,E2 416.1856} C_DIS
LIN {X 111.3434,Y 80.3904,Z 175,A 37.4961,B 7.6182,C 0.1578,E1 7.7491,E2 414.372} C_DIS
LIN {X 108.7409,Y 83.8775,Z 175,A 39.3074,B 7.6182,C 0.1537,E1 7.7461,E2 412.5605} C_DIS
LIN {X 105.9791,Y 87.341,Z 175,A 41.0121,B 7.6183,C 0.1523,E1 7.7431,E2 410.8731} C_DIS
LIN {X 103.2643,Y 90.5345,Z 175,A 42.7809,B 7.6184,C 0.1482,E1 7.7399,E2 409.1011} C_DIS
LIN {X 100.7212,Y 93.3555,Z 175,A 44.2989,B 7.6184,C 0.1461,E1 7.737,E2 407.591} C_DIS
LIN {X 98.2713,Y 95.931,Z 175,A 45.8795,B 7.6185,C 0.1412,E1 7.7339,E2 405.9977} C_DIS
LIN {X 95.2049,Y 98.9755,Z 175,A 47.5408,B 7.6185,C 0.1402,E1 7.7306,E2 404.3535} C_DIS
LIN {X 92.6117,Y 101.4061,Z 175,A 49.1186,B 7.6186,C 0.1356,E1 7.7274,E2 402.7635} C_DIS
LIN {X 89.2855,Y 104.3466,Z 175,A 50.932,B 7.6186,C 0.1328,E1 7.7236,E2 400.9546} C_DIS
LIN {X 85.8703,Y 107.1746,Z 175,A 52.7791,B 7.6187,C 0.1295,E1 7.7196,E2 399.1075} C_DIS
LIN {X 82.3719,Y 109.8862,Z 175,A 54.602,B 7.6187,C 0.1268,E1 7.7155,E2 397.2872} C_DIS
LIN {X 78.6963,Y 112.5474,Z 175,A 56.4739,B 7.6188,C 0.124,E1 7.7113,E2 395.4178} C_DIS
LIN {X 74.9925,Y 115.0483,Z 175,A 58.3093,B 7.6188,C 0.1216,E1 7.707,E2 393.5858} C_DIS
LIN {X 71.3344,Y 117.3517,Z 175,A 60.1015,B 7.6189,C 0.1191,E1 7.7027,E2 391.795} C_DIS
LIN {X 67.6679,Y 119.5038,Z 175,A 61.8085,B 7.6189,C 0.1178,E1 7.6986,E2 390.0962} C_DIS
LIN {X 64.2636,Y 121.3663,Z 175,A 63.1986,B 7.6189,C 0.1197,E1 7.6953,E2 388.7344} C_DIS
LIN {X 61.3163,Y 122.8823,Z 175,A 64.7135,B 7.6189,C 0.1155,E1 7.6915,E2 387.2031} C_DIS
LIN {X 57.9909,Y 124.4852,Z 175,A 66.1575,B 7.6189,C 0.1154,E1 7.6879,E2 385.7711} C_DIS
LIN {X 54.8837,Y 125.8862,Z 175,A 67.5864,B 7.6189,C 0.1136,E1 7.6842,E2 384.3415} C_DIS
LIN {X 51.9156,Y 127.1398,Z 175,A 68.896,B 7.619,C 0.1127,E1 7.6808,E2 383.0363} C_DIS
LIN {X 48.9646,Y 128.3066,Z 175,A 70.3715,B 7.619,C 0.1087,E1 7.6769,E2 381.5422} C_DIS
LIN {X 45.3436,Y 129.6283,Z 175,A 71.8822,B 7.619,C 0.1088,E1 7.673,E2 380.0438} C_DIS
LIN {X 42.2251,Y 130.6777,Z 175,A 73.2107,B 7.619,C 0.1084,E1 7.6695,E2 378.7209} C_DIS
LIN {X 39.1683,Y 131.6268,Z 175,A 74.5804,B 7.619,C 0.1067,E1 7.6658,E2 377.3473} C_DIS
LIN {X 35.9649,Y 132.5379,Z 175,A 76.0108,B 7.6191,C 0.1049,E1 7.662,E2 375.9121} C_DIS
LIN {X 32.7749,Y 133.3627,Z 175,A 77.249,B 7.6191,C 0.1063,E1 7.6587,E2 374.6911} C_DIS
LIN {X 29.3569,Y 134.1557,Z 175,A 78.6231,B 7.6191,C 0.1069,E1 7.6549,E2 373.3284} C_DIS
LIN {X 26.3643,Y 134.7766,Z 175,A 80.1238,B 7.6191,C 0.1023,E1 7.6508,E2 371.8003} C_DIS
LIN {X 22.9736,Y 135.395,Z 175,A 81.4929,B 7.6191,C 0.1028,E1 7.647,E2 370.44} C_DIS
LIN {X 20.0004,Y 135.8668,Z 175,A 82.7321,B 7.6191,C 0.1025,E1 7.6436,E2 369.2034} C_DIS
LIN {X 16.8375,Y 136.2949,Z 175,A 84.1587,B 7.6191,C 0.1004,E1 7.6396,E2 367.7654} C_DIS
LIN {X 13.6907,Y 136.6469,Z 175,A 85.2946,B 7.6191,C 0.1031,E1 7.6365,E2 366.6529} C_DIS
LIN {X 10.5624,Y 136.9243,Z 175,A 86.6801,B 7.6191,C 0.1016,E1 7.6326,E2 365.2586} C_DIS
LIN {X 7.6684,Y 137.1179,Z 175,A 87.9561,B 7.6191,C 0.1003,E1 7.6291,E2 363.9749} C_DIS
LIN {X 4.5821,Y 137.2557,Z 175,A 89.2411,B 7.6191,C 0.1003,E1 7.6255,E2 362.691} C_DIS
LIN {X 1.0985,Y 137.326,Z 175,A 90.6357,B 7.6191,C 0.1011,E1 7.6216,E2 361.3043} C_DIS
LIN {X -3.26,Y 137.2924,Z 175,A 92.3658,B 7.6191,C 0.1026,E1 7.6168,E2 359.5859} C_DIS
LIN {X -6.3358,Y 137.1849,Z 175,A 93.6528,B 7.6191,C 0.1027,E1 7.6132,E2 358.2992} C_DIS
LIN {X -9.2202,Y 137.0223,Z 175,A 95.0125,B 7.6191,C 0.1005,E1 7.6094,E2 356.9211} C_DIS
LIN {X -12.3399,Y 136.7766,Z 175,A 96.2515,B 7.6191,C 0.1019,E1 7.606,E2 355.6911} C_DIS
LIN {X -15.4791,Y 136.457,Z 175,A 97.5734,B 7.6191,C 0.1022,E1 7.6023,E2 354.3691} C_DIS
LIN {X -19.0976,Y 135.9958,Z 175,A 99.0254,B 7.6191,C 0.1039,E1 7.5983,E2 352.9265} C_DIS
LIN {X -22.0259,Y 135.5532,Z 175,A 100.3436,B 7.6191,C 0.1031,E1 7.5946,E2 351.5989} C_DIS
LIN {X -24.9894,Y 135.0394,Z 175,A 101.6783,B 7.6191,C 0.1025,E1 7.5909,E2 350.2552} C_DIS
LIN {X -28.1819,Y 134.4094,Z 175,A 103.0441,B 7.6191,C 0.1032,E1 7.5872,E2 348.8892} C_DIS
LIN {X -31.6743,Y 133.628,Z 175,A 104.4481,B 7.6191,C 0.1055,E1 7.5834,E2 347.4971} C_DIS
LIN {X -34.5841,Y 132.9062,Z 175,A 105.7303,B 7.6191,C 0.1059,E1 7.5799,E2 346.2119} C_DIS
LIN {X -37.9297,Y 131.9895,Z 175,A 107.2918,B 7.6191,C 0.1053,E1 7.5757,E2 344.6372} C_DIS
LIN {X -41.2199,Y 130.9988,Z 175,A 108.6283,B 7.6191,C 0.108,E1 7.5722,E2 343.3137} C_DIS
LIN {X -44.1864,Y 130.0295,Z 175,A 109.943,B 7.6191,C 0.109,E1 7.5687,E2 341.9984} C_DIS
LIN {X -47.5942,Y 128.8199,Z 175,A 111.4639,B 7.6191,C 0.1103,E1 7.5647,E2 340.477} C_DIS
LIN {X -50.5512,Y 127.6898,Z 175,A 112.7952,B 7.6191,C 0.1115,E1 7.5612,E2 339.1453} C_DIS
LIN {X -53.713,Y 126.3924,Z 175,A 114.3593,B 7.6191,C 0.111,E1 7.5572,E2 337.5653} C_DIS
LIN {X -57.0504,Y 124.9201,Z 175,A 115.6891,B 7.619,C 0.1157,E1 7.5538,E2 336.2603} C_DIS
LIN {X -59.9786,Y 123.5422,Z 175,A 117.2111,B 7.619,C 0.1148,E1 7.5499,E2 334.7181} C_DIS
LIN {X -63.2883,Y 121.8784,Z 175,A 118.7519,B 7.619,C 0.1169,E1 7.5461,E2 333.1791} C_DIS
LIN {X -67.0124,Y 119.8722,Z 175,A 120.578,B 7.619,C 0.1185,E1 7.5416,E2 331.347} C_DIS
LIN {X -70.6883,Y 117.7424,Z 175,A 122.2673,B 7.6189,C 0.1223,E1 7.5376,E2 329.6694} C_DIS
LIN {X -73.6723,Y 115.8987,Z 175,A 123.7789,B 7.6189,C 0.1239,E1 7.534,E2 328.153} C_DIS
LIN {X -77.077,Y 113.662,Z 175,A 125.5108,B 7.6189,C 0.1261,E1 7.53,E2 326.4185} C_DIS
LIN {X -80.3342,Y 111.3842,Z 175,A 127.2639,B 7.6188,C 0.1275,E1 7.526,E2 324.6552} C_DIS
LIN {X -83.919,Y 108.7088,Z 175,A 129.1415,B 7.6188,C 0.1306,E1 7.5218,E2 322.7778} C_DIS
LIN {X -87.341,Y 105.9791,Z 175,A 130.9892,B 7.6187,C 0.1337,E1 7.5178,E2 320.9292} C_DIS
LIN {X -90.6269,Y 103.1837,Z 175,A 132.7386,B 7.6186,C 0.1378,E1 7.5141,E2 319.1877} C_DIS
LIN {X -93.3555,Y 100.7212,Z 175,A 134.2603,B 7.6186,C 0.141,E1 7.511,E2 317.6688} C_DIS
LIN {X -95.931,Y 98.2713,Z 175,A 135.8851,B 7.6186,C 0.1419,E1 7.5077,E2 316.0278} C_DIS
LIN {X -99.0034,Y 95.1756,Z 175,A 137.5978,B 7.6184,C 0.1472,E1 7.5044,E2 314.33} C_DIS
LIN {X -101.4061,Y 92.6117,Z 175,A 139.1286,B 7.6184,C 0.1494,E1 7.5015,E2 312.7925} C_DIS
LIN {X -104.2666,Y 89.3783,Z 175,A 140.9376,B 7.6184,C 0.1532,E1 7.4981,E2 310.9843} C_DIS
LIN {X -106.6182,Y 86.5602,Z 175,A 142.5105,B 7.6182,C 0.1561,E1 7.4953,E2 309.4077} C_DIS
LIN {X -108.9246,Y 83.6386,Z 175,A 144.1621,B 7.6182,C 0.1583,E1 7.4925,E2 307.7454} C_DIS
LIN {X -111.4558,Y 80.2354,Z 175,A 145.8841,B 7.6182,C 0.1631,E1 7.4897,E2 306.0309} C_DIS
LIN {X -113.9057,Y 76.7171,Z 175,A 147.7187,B 7.618,C 0.1667,E1 7.4868,E2 304.1924} C_DIS
LIN {X -115.9634,Y 73.5697,Z 175,A 149.3826,B 7.618,C 0.1692,E1 7.4842,E2 302.5182} C_DIS
LIN {X -118.1905,Y 69.9365,Z 175,A 151.0696,B 7.6178,C 0.1749,E1 7.4818,E2 300.8442} C_DIS
LIN {X -119.9896,Y 66.8021,Z 175,A 152.7213,B 7.6178,C 0.1767,E1 7.4795,E2 299.1761} C_DIS
LIN {X -122.0534,Y 62.9511,Z 175,A 154.4881,B 7.6177,C 0.1821,E1 7.4773,E2 297.4181} C_DIS
LIN {X -123.645,Y 59.7635,Z 175,A 155.9669,B 7.6176,C 0.1861,E1 7.4754,E2 295.9416} C_DIS
LIN {X -125.0098,Y 56.8566,Z 175,A 157.4084,B 7.6176,C 0.1882,E1 7.4737,E2 294.4889} C_DIS
LIN {X -126.4834,Y 53.4949,Z 175,A 158.9645,B 7.6174,C 0.192,E1 7.472,E2 292.9311} C_DIS
LIN {X -127.6898,Y 50.5512,Z 175,A 160.2374,B 7.6174,C 0.1963,E1 7.4707,E2 291.6663} C_DIS
LIN {X -128.9814,Y 47.1547,Z 175,A 161.7793,B 7.6172,C 0.2,E1 7.4692,E2 290.1227} C_DIS
LIN {X -130.0295,Y 44.1864,Z 175,A 163.2434,B 7.6172,C 0.2016,E1 7.4679,E2 288.6411} C_DIS
LIN {X -131.2074,Y 40.5485,Z 175,A 164.6659,B 7.617,C 0.2083,E1 7.4667,E2 287.2415} C_DIS
LIN {X -132.0928,Y 37.5668,Z 175,A 166.0595,B 7.617,C 0.2106,E1 7.4656,E2 285.8372} C_DIS
LIN {X -132.9062,Y 34.5841,Z 175,A 167.3726,B 7.6169,C 0.2139,E1 7.4647,E2 284.5226} C_DIS
LIN {X -133.6987,Y 31.3811,Z 175,A 168.9179,B 7.6169,C 0.2155,E1 7.4636,E2 282.9574} C_DIS
LIN {X -134.4094,Y 28.1819,Z 175,A 170.2394,B 7.6167,C 0.22,E1 7.4629,E2 281.643} C_DIS
LIN {X -135.0394,Y 24.9894,Z 175,A 171.5469,B 7.6165,C 0.2245,E1 7.4622,E2 280.343} C_DIS
LIN {X -135.6137,Y 21.6521,Z 175,A 173.1033,B 7.6165,C 0.2266,E1 7.4615,E2 278.7699} C_DIS
LIN {X -136.0992,Y 18.3504,Z 175,A 174.38,B 7.6163,C 0.2322,E1 7.461,E2 277.509} C_DIS
LIN {X -136.5191,Y 14.9019,Z 175,A 175.7646,B 7.6162,C 0.2372,E1 7.4605,E2 276.1338} C_DIS
LIN {X -136.7766,Y 12.3399,Z 175,A 177.0421,B 7.6162,C 0.2375,E1 7.4602,E2 274.8319} C_DIS
LIN {X -137.0355,Y 9.0059,Z 175,A 178.3096,B 7.616,C 0.2433,E1 7.4599,E2 273.5816} C_DIS
LIN {X -137.2162,Y 5.5947,Z 175,A 179.8922,B 7.616,C 0.2452,E1 7.4597,E2 271.9805} C_DIS
LIN {X -137.3161,Y 1.9761,Z 175,A -178.6015,B 7.6158,C 0.2496,E1 7.4597,E2 270.4761} C_DIS
LIN {X -137.3237,Y -1.5208,Z 175,A -177.0625,B 7.6157,C 0.2528,E1 7.4597,E2 268.9283} C_DIS
LIN {X -137.2557,Y -4.5821,Z 175,A -175.7565,B 7.6156,C 0.2561,E1 7.4597,E2 267.6199} C_DIS
LIN {X -137.0793,Y -8.2939,Z 175,A -174.3118,B 7.6154,C 0.2619,E1 7.46,E2 266.1896} C_DIS
LIN {X -136.8867,Y -11.0366,Z 175,A -173.0031,B 7.6154,C 0.263,E1 7.4603,E2 264.8617} C_DIS
LIN {X -136.6261,Y -13.9072,Z 175,A -171.8436,B 7.6152,C 0.2671,E1 7.4606,E2 263.7086} C_DIS
LIN {X -136.269,Y -17.0552,Z 175,A -170.4935,B 7.6151,C 0.2704,E1 7.461,E2 262.356} C_DIS
LIN {X -135.7975,Y -20.4647,Z 175,A -169.0266,B 7.6149,C 0.2741,E1 7.4616,E2 260.8863} C_DIS
LIN {X -135.2851,Y -23.6165,Z 175,A -167.7039,B 7.6148,C 0.278,E1 7.4622,E2 259.5659} C_DIS
LIN {X -134.6896,Y -26.8052,Z 175,A -166.2871,B 7.6147,C 0.2809,E1 7.463,E2 258.1421} C_DIS
LIN {X -134.0137,Y -30.0018,Z 175,A -164.8933,B 7.6146,C 0.2843,E1 7.4638,E2 256.7455} C_DIS
LIN {X -133.2566,Y -33.2035,Z 175,A -163.5793,B 7.6144,C 0.289,E1 7.4647,E2 255.4399} C_DIS
LIN {X -132.4789,Y -36.1862,Z 175,A -162.1807,B 7.6144,C 0.291,E1 7.4657,E2 254.028} C_DIS
LIN {X -131.4944,Y -39.6104,Z 175,A -160.5975,B 7.6142,C 0.2937,E1 7.467,E2 252.4336} C_DIS
LIN {X -130.3791,Y -43.1365,Z 175,A -159.1218,B 7.614,C 0.2988,E1 7.4682,E2 250.9674} C_DIS
LIN {X -129.4764,Y -45.7818,Z 175,A -157.8234,B 7.614,C 0.3001,E1 7.4694,E2 249.6531} C_DIS
LIN {X -128.2214,Y -49.1837,Z 175,A -156.4482,B 7.6137,C 0.3061,E1 7.4708,E2 248.2963} C_DIS
LIN {X -127.0517,Y -52.1342,Z 175,A -155.0032,B 7.6137,C 0.3079,E1 7.4723,E2 246.8369} C_DIS
LIN {X -125.6148,Y -55.504,Z 175,A -153.5422,B 7.6135,C 0.3128,E1 7.4739,E2 245.3853} C_DIS
LIN {X -124.2866,Y -58.4205,Z 175,A -151.9859,B 7.6135,C 0.3132,E1 7.4758,E2 243.8021} C_DIS
LIN {X -122.603,Y -61.8717,Z 175,A -150.5049,B 7.6132,C 0.319,E1 7.4776,E2 242.3372} C_DIS
LIN {X -121.1253,Y -64.72,Z 175,A -148.9773,B 7.6132,C 0.3197,E1 7.4796,E2 240.7865} C_DIS
LIN {X -119.0108,Y -68.5307,Z 175,A -147.2459,B 7.6129,C 0.3254,E1 7.482,E2 239.067} C_DIS
LIN {X -117.0955,Y -71.7536,Z 175,A -145.575,B 7.6129,C 0.3276,E1 7.4844,E2 237.3834} C_DIS
LIN {X -114.8796,Y -75.2509,Z 175,A -143.8287,B 7.6127,C 0.3314,E1 7.487,E2 235.6355} C_DIS
LIN {X -112.4379,Y -78.8529,Z 175,A -141.9522,B 7.6125,C 0.3348,E1 7.49,E2 233.752} C_DIS
LIN {X -109.8862,Y -82.3719,Z 175,A -140.1787,B 7.6123,C 0.3394,E1 7.493,E2 231.9844} C_DIS
LIN {X -107.2508,Y -85.7746,Z 175,A -138.3157,B 7.6122,C 0.3424,E1 7.4962,E2 230.1135} C_DIS
LIN {X -104.4941,Y -89.112,Z 175,A -136.5261,B 7.612,C 0.3465,E1 7.4994,E2 228.3267} C_DIS
LIN {X -101.9205,Y -92.0447,Z 175,A -134.9035,B 7.6118,C 0.35,E1 7.5024,E2 226.7053} C_DIS
LIN {X -99.5047,Y -94.6511,Z 175,A -133.3061,B 7.6118,C 0.3513,E1 7.5055,E2 225.0937} C_DIS
LIN {X -96.4779,Y -97.7349,Z 175,A -131.5735,B 7.6116,C 0.3559,E1 7.5089,E2 223.3706} C_DIS
LIN {X -93.8754,Y -100.2371,Z 175,A -130.0631,B 7.6114,C 0.3587,E1 7.5119,E2 221.86} C_DIS
LIN {X -90.9819,Y -102.8699,Z 175,A -128.323,B 7.6114,C 0.3601,E1 7.5156,E2 220.1065} C_DIS
LIN {X -87.9298,Y -105.4916,Z 175,A -126.5785,B 7.6113,C 0.3621,E1 7.5193,E2 218.3539} C_DIS
LIN {X -84.4806,Y -108.2734,Z 175,A -124.7168,B 7.6111,C 0.3651,E1 7.5234,E2 216.4909} C_DIS
LIN {X -80.9506,Y -110.9374,Z 175,A -122.9306,B 7.611,C 0.369,E1 7.5274,E2 214.7125} C_DIS
LIN {X -77.972,Y -113.0503,Z 175,A -121.3045,B 7.611,C 0.3698,E1 7.5312,E2 213.0734} C_DIS
LIN {X -74.2175,Y -115.5496,Z 175,A -119.551,B 7.6107,C 0.3745,E1 7.5352,E2 211.3366} C_DIS
LIN {X -71.3344,Y -117.3517,Z 175,A -117.9745,B 7.6107,C 0.3741,E1 7.539,E2 209.7399} C_DIS
LIN {X -67.6058,Y -119.5387,Z 175,A -116.1448,B 7.6107,C 0.3761,E1 7.5435,E2 207.9068} C_DIS
LIN {X -64.6142,Y -121.1822,Z 175,A -114.839,B 7.6104,C 0.3797,E1 7.5466,E2 206.6163} C_DIS
LIN {X -61.3163,Y -122.8823,Z 175,A -113.2106,B 7.6104,C 0.3803,E1 7.5507,E2 204.9774} C_DIS
LIN {X -57.939,Y -124.5092,Z 175,A -111.9029,B 7.6101,C 0.3861,E1 7.5539,E2 203.7026} C_DIS
LIN {X -55.0698,Y -125.8057,Z 175,A -110.384,B 7.6101,C 0.3843,E1 7.5579,E2 202.1573} C_DIS
LIN {X -51.9156,Y -127.1398,Z 175,A -109.0343,B 7.6101,C 0.387,E1 7.5613,E2 200.8176} C_DIS
LIN {X -48.9646,Y -128.3066,Z 175,A -107.47,B 7.6101,C 0.3844,E1 7.5655,E2 199.2221} C_DIS
LIN {X -45.4665,Y -129.5857,Z 175,A -106.0684,B 7.6101,C 0.3882,E1 7.5691,E2 197.84} C_DIS
LIN {X -42.589,Y -130.5614,Z 175,A -104.7821,B 7.61,C 0.3889,E1 7.5725,E2 196.551} C_DIS
LIN {X -39.1683,Y -131.6268,Z 175,A -103.1952,B 7.61,C 0.3885,E1 7.5768,E2 194.952} C_DIS
LIN {X -35.9649,Y -132.5379,Z 175,A -101.9731,B 7.6098,C 0.3921,E1 7.58,E2 193.7511} C_DIS
LIN {X -32.629,Y -133.3979,Z 175,A -100.5822,B 7.6098,C 0.3937,E1 7.5838,E2 192.3658} C_DIS
LIN {X -29.56,Y -134.1119,Z 175,A -99.214,B 7.6098,C 0.3935,E1 7.5875,E2 190.9904} C_DIS
LIN {X -26.097,Y -134.8277,Z 175,A -97.6213,B 7.6098,C 0.3922,E1 7.5919,E2 189.3821} C_DIS
LIN {X -21.8063,Y -135.5898,Z 175,A -95.7613,B 7.6098,C 0.3922,E1 7.5971,E2 187.5163} C_DIS
LIN {X -18.4171,Y -136.0905,Z 175,A -94.4038,B 7.6098,C 0.3938,E1 7.6008,E2 186.1675} C_DIS
LIN {X -15.262,Y -136.4804,Z 175,A -92.9723,B 7.6098,C 0.3923,E1 7.6048,E2 184.7219} C_DIS
LIN {X -12.3399,Y -136.7766,Z 175,A -91.7834,B 7.6098,C 0.3931,E1 7.6081,E2 183.5373} C_DIS
LIN {X -9.0059,Y -137.0355,Z 175,A -90.539,B 7.6096,C 0.3958,E1 7.6115,E2 182.3118} C_DIS
LIN {X -5.9096,Y -137.2039,Z 175,A -89.2468,B 7.6096,C 0.3958,E1 7.6151,E2 181.0193} C_DIS
LIN {X -2.8373,Y -137.3018,Z 175,A -87.7846,B 7.6098,C 0.3927,E1 7.6193,E2 179.5332} C_DIS
LIN {X 1.0205,Y -137.3262,Z 175,A -86.614,B 7.6094,C 0.4001,E1 7.6224,E2 178.4185} C_DIS
Enddeposition()
LIN {X 1.0205,Y -137.3262,Z 175,A -86.614,B 7.6094,C 0.4001,E1 7.6224,E2 178.4185} C_DIS
Startdeposition()
$VEL.CP = VEL_PRINT
LIN {X -0.7055,Y -138.2347,Z 175,A -87.5582,B 7.5596,C 0.4088,E1 7.5703,E2 179.4403} C_DIS
LIN {X -4.7394,Y -138.1567,Z 175,A -89.3291,B 7.5596,C 0.4105,E1 7.5653,E2 181.2247} C_DIS
LIN {X -9.3349,Y -137.9228,Z 175,A -91.1751,B 7.5596,C 0.4094,E1 7.5602,E2 183.0636} C_DIS
LIN {X -13.1495,Y -137.6095,Z 175,A -92.71,B 7.5596,C 0.4083,E1 7.5559,E2 184.5925} C_DIS
LIN {X -16.2919,Y -137.2729,Z 175,A -93.9295,B 7.5597,C 0.4066,E1 7.5526,E2 185.8007} C_DIS
LIN {X -18.8106,Y -136.9525,Z 175,A -95.0399,B 7.5597,C 0.4073,E1 7.5495,E2 186.9191} C_DIS
LIN {X -25.2552,Y -135.9115,Z 175,A -97.8984,B 7.5597,C 0.4088,E1 7.5416,E2 189.7982} C_DIS
LIN {X -32.3123,Y -134.4067,Z 175,A -100.6251,B 7.5599,C 0.403,E1 7.5342,E2 192.4917} C_DIS
LIN {X -35.458,Y -133.6113,Z 175,A -102.2837,B 7.5597,C 0.4073,E1 7.5296,E2 194.191} C_DIS
LIN {X -39.9244,Y -132.3464,Z 175,A -104.0523,B 7.5599,C 0.4035,E1 7.5249,E2 195.94} C_DIS
LIN {X -43.3829,Y -131.2525,Z 175,A -105.5384,B 7.5599,C 0.402,E1 7.521,E2 197.4241} C_DIS
LIN {X -46.6386,Y -130.1311,Z 175,A -107.0354,B 7.5599,C 0.402,E1 7.517,E2 198.9304} C_DIS
LIN {X -49.8825,Y -128.9223,Z 175,A -108.3992,B 7.5601,C 0.3995,E1 7.5135,E2 200.2852} C_DIS
LIN {X -52.999,Y -127.6729,Z 175,A -109.8738,B 7.5601,C 0.3995,E1 7.5096,E2 201.7706} C_DIS
LIN {X -55.8464,Y -126.4546,Z 175,A -111.2936,B 7.5601,C 0.4002,E1 7.5059,E2 203.208} C_DIS
LIN {X -59.2869,Y -124.8773,Z 175,A -112.7448,B 7.5603,C 0.3967,E1 7.5023,E2 204.6442} C_DIS
LIN {X -61.9643,Y -123.573,Z 175,A -114.0563,B 7.5603,C 0.3964,E1 7.499,E2 205.9657} C_DIS
LIN {X -66.9016,Y -120.9707,Z 175,A -116.3982,B 7.5604,C 0.3939,E1 7.4932,E2 208.3113} C_DIS
LIN {X -70.7359,Y -118.7693,Z 175,A -118.2115,B 7.5606,C 0.3912,E1 7.4889,E2 210.1221} C_DIS
LIN {X -73.3983,Y -117.1434,Z 175,A -119.6481,B 7.5606,C 0.3915,E1 7.4854,E2 211.577} C_DIS
LIN {X -77.5399,Y -114.4434,Z 175,A -121.5987,B 7.5608,C 0.3869,E1 7.4809,E2 213.5148} C_DIS
LIN {X -82.9392,Y -110.5937,Z 175,A -124.4516,B 7.5609,C 0.3841,E1 7.4744,E2 216.3807} C_DIS
LIN {X -86.5974,Y -107.7528,Z 175,A -126.3325,B 7.5611,C 0.3803,E1 7.4703,E2 218.2563} C_DIS
LIN {X -89.9305,Y -104.9874,Z 175,A -128.214,B 7.5611,C 0.3784,E1 7.4663,E2 220.1485} C_DIS
LIN {X -93.2938,Y -102.0103,Z 175,A -130.0974,B 7.5614,C 0.3753,E1 7.4624,E2 222.0342} C_DIS
LIN {X -96.6928,Y -98.7939,Z 175,A -132.1414,B 7.5614,C 0.3731,E1 7.4582,E2 224.091} C_DIS
LIN {X -100.3106,Y -95.119,Z 175,A -134.2073,B 7.5617,C 0.3677,E1 7.4542,E2 226.1471} C_DIS
LIN {X -104.3682,Y -90.6482,Z 175,A -136.7333,B 7.562,C 0.3629,E1 7.4495,E2 228.6752} C_DIS
LIN {X -107.2755,Y -87.1884,Z 175,A -138.637,B 7.5621,C 0.3593,E1 7.4461,E2 230.5822} C_DIS
LIN {X -110.0776,Y -83.6231,Z 175,A -140.5756,B 7.5623,C 0.356,E1 7.4428,E2 232.5275} C_DIS
LIN {X -112.7725,Y -79.9512,Z 175,A -142.49,B 7.5625,C 0.352,E1 7.4397,E2 234.4444} C_DIS
LIN {X -115.3963,Y -76.1146,Z 175,A -144.4096,B 7.5627,C 0.3474,E1 7.4367,E2 236.3623} C_DIS
LIN {X -117.8148,Y -72.3145,Z 175,A -146.2715,B 7.5629,C 0.3429,E1 7.4339,E2 238.2226} C_DIS
LIN {X -119.8311,Y -68.9229,Z 175,A -147.9626,B 7.563,C 0.3397,E1 7.4315,E2 239.9199} C_DIS
LIN {X -122.8629,Y -63.3592,Z 175,A -150.6673,B 7.5633,C 0.3342,E1 7.428,E2 242.6331} C_DIS
LIN {X -124.5687,Y -59.9328,Z 175,A -152.1184,B 7.5635,C 0.3283,E1 7.4262,E2 244.0661} C_DIS
LIN {X -126.2511,Y -56.3014,Z 175,A -153.8632,B 7.5637,C 0.3252,E1 7.4242,E2 245.8208} C_DIS
LIN {X -127.6853,Y -52.9694,Z 175,A -155.3387,B 7.5638,C 0.3209,E1 7.4226,E2 247.2919} C_DIS
LIN {X -129.1605,Y -49.2692,Z 175,A -157.1073,B 7.564,C 0.3181,E1 7.4208,E2 249.0744} C_DIS
LIN {X -130.8284,Y -44.6495,Z 175,A -159.2786,B 7.5641,C 0.3145,E1 7.4187,E2 251.2614} C_DIS
LIN {X -132.108,Y -40.7031,Z 175,A -160.6655,B 7.5645,C 0.3053,E1 7.4176,E2 252.605} C_DIS
LIN {X -133.0636,Y -37.4614,Z 175,A -162.337,B 7.5645,C 0.3051,E1 7.4163,E2 254.3097} C_DIS
LIN {X -133.8316,Y -34.6227,Z 175,A -163.654,B 7.5645,C 0.3031,E1 7.4153,E2 255.6383} C_DIS
LIN {X -134.7298,Y -30.9375,Z 175,A -165.1244,B 7.5648,C 0.2973,E1 7.4144,E2 257.0947} C_DIS
LIN {X -135.4383,Y -27.6719,Z 175,A -166.5814,B 7.5649,C 0.2944,E1 7.4135,E2 258.5597} C_DIS
LIN {X -136.1054,Y -24.1786,Z 175,A -168.0936,B 7.5651,C 0.2908,E1 7.4128,E2 260.0756} C_DIS
LIN {X -136.6964,Y -20.5836,Z 175,A -169.7281,B 7.5651,C 0.2882,E1 7.412,E2 261.7245} C_DIS
LIN {X -137.2044,Y -16.8665,Z 175,A -171.065,B 7.5654,C 0.2808,E1 7.4116,E2 263.0327} C_DIS
LIN {X -137.6461,Y -12.7683,Z 175,A -173.064,B 7.5654,C 0.2799,E1 7.411,E2 265.0668} C_DIS
LIN {X -137.9736,Y -8.5208,Z 175,A -174.6295,B 7.5657,C 0.2721,E1 7.4107,E2 266.6057} C_DIS
LIN {X -138.1379,Y -5.2216,Z 175,A -176.1428,B 7.5658,C 0.2701,E1 7.4105,E2 268.136} C_DIS
LIN {X -138.2325,Y -1.1931,Z 175,A -178.0218,B 7.5658,C 0.2681,E1 7.4105,E2 270.0397} C_DIS
LIN {X -138.1897,Y 3.6042,Z 175,A -179.8836,B 7.5661,C 0.2607,E1 7.4105,E2 271.8839} C_DIS
LIN {X -138.0438,Y 7.3042,Z 175,A 178.5422,B 7.5663,C 0.2568,E1 7.4107,E2 273.4617} C_DIS
LIN {X -137.854,Y 10.2778,Z 175,A 177.1469,B 7.5663,C 0.2554,E1 7.411,E2 274.8758} C_DIS
LIN {X -137.3626,Y 15.5361,Z 175,A 174.9423,B 7.5665,C 0.2493,E1 7.4116,E2 277.0804} C_DIS
LIN {X -136.84,Y 19.5978,Z 175,A 173.4331,B 7.5668,C 0.2419,E1 7.4122,E2 278.5646} C_DIS
LIN {X -135.9153,Y 25.2352,Z 175,A 170.5907,B 7.5668,C 0.2415,E1 7.4135,E2 281.4638} C_DIS
LIN {X -135.2456,Y 28.6042,Z 175,A 169.3853,B 7.567,C 0.2346,E1 7.4142,E2 282.6409} C_DIS
LIN {X -134.4423,Y 32.1643,Z 175,A 168.0459,B 7.5672,C 0.228,E1 7.415,E2 283.9572} C_DIS
LIN {X -133.5866,Y 35.5506,Z 175,A 166.4793,B 7.5672,C 0.2256,E1 7.4161,E2 285.5373} C_DIS
LIN {X -132.6886,Y 38.7679,Z 175,A 165.0238,B 7.5673,C 0.2227,E1 7.4173,E2 287.0003} C_DIS
LIN {X -131.6602,Y 42.1283,Z 175,A 163.5763,B 7.5675,C 0.2185,E1 7.4185,E2 288.4453} C_DIS
LIN {X -130.6294,Y 45.2234,Z 175,A 162.3717,B 7.5676,C 0.2128,E1 7.4195,E2 289.6302} C_DIS
LIN {X -129.8237,Y 47.4912,Z 175,A 161.179,B 7.5676,C 0.2128,E1 7.4207,E2 290.8463} C_DIS
LIN {X -128.3875,Y 51.2449,Z 175,A 159.4729,B 7.5677,C 0.2088,E1 7.4224,E2 292.5557} C_DIS
LIN {X -126.8885,Y 54.8496,Z 175,A 157.8581,B 7.5679,C 0.2044,E1 7.4242,E2 294.1685} C_DIS
LIN {X -125.7117,Y 57.4984,Z 175,A 156.7066,B 7.5679,C 0.2006,E1 7.4255,E2 295.3127} C_DIS
LIN {X -124.3888,Y 60.3095,Z 175,A 155.005,B 7.5679,C 0.2028,E1 7.4276,E2 297.0642} C_DIS
LIN {X -122.0361,Y 64.9378,Z 175,A 153.0556,B 7.5681,C 0.1946,E1 7.4301,E2 298.9866} C_DIS
LIN {X -119.9266,Y 68.7563,Z 175,A 151.2444,B 7.5682,C 0.1901,E1 7.4325,E2 300.7964} C_DIS
LIN {X -117.8575,Y 72.245,Z 175,A 149.6504,B 7.5684,C 0.1847,E1 7.4348,E2 302.378} C_DIS
LIN {X -115.7801,Y 75.53,Z 175,A 147.8352,B 7.5684,C 0.1836,E1 7.4376,E2 304.2169} C_DIS
LIN {X -113.4768,Y 78.9476,Z 175,A 146.0994,B 7.5684,C 0.1799,E1 7.4403,E2 305.9545} C_DIS
LIN {X -111.1385,Y 82.2071,Z 175,A 144.1772,B 7.5684,C 0.1795,E1 7.4435,E2 307.907} C_DIS
LIN {X -109.1093,Y 84.8818,Z 175,A 143.0122,B 7.5686,C 0.1732,E1 7.4455,E2 309.0429} C_DIS
LIN {X -106.582,Y 88.0342,Z 175,A 141.3063,B 7.5687,C 0.1699,E1 7.4485,E2 310.7509} C_DIS
LIN {X -103.8873,Y 91.1993,Z 175,A 139.5139,B 7.5687,C 0.1671,E1 7.4518,E2 312.5503} C_DIS
LIN {X -100.657,Y 94.7518,Z 175,A 137.5032,B 7.5689,C 0.1631,E1 7.4556,E2 314.5617} C_DIS
LIN {X -97.6387,Y 97.8595,Z 175,A 135.6555,B 7.5689,C 0.1602,E1 7.4592,E2 316.4141} C_DIS
LIN {X -94.512,Y 100.8829,Z 175,A 133.8533,B 7.5689,C 0.1566,E1 7.4629,E2 318.2146} C_DIS
LIN {X -91.0469,Y 104.0203,Z 175,A 131.8903,B 7.5691,C 0.1532,E1 7.467,E2 320.179} C_DIS
LIN {X -87.5846,Y 106.9517,Z 175,A 130.0388,B 7.5691,C 0.1493,E1 7.4709,E2 322.0252} C_DIS
LIN {X -84.545,Y 109.3704,Z 175,A 128.1481,B 7.5691,C 0.1504,E1 7.4752,E2 323.9489} C_DIS
LIN {X -81.8613,Y 111.3932,Z 175,A 126.977,B 7.5692,C 0.1449,E1 7.4777,E2 325.0916} C_DIS
LIN {X -78.4291,Y 113.8361,Z 175,A 125.168,B 7.5692,C 0.1429,E1 7.4819,E2 326.9068} C_DIS
LIN {X -74.7757,Y 116.2686,Z 175,A 123.2795,B 7.5692,C 0.141,E1 7.4863,E2 328.8024} C_DIS
LIN {X -70.5063,Y 118.9062,Z 175,A 120.9618,B 7.5692,C 0.1414,E1 7.4919,E2 331.1474} C_DIS
LIN {X -67.2519,Y 120.7767,Z 175,A 119.6385,B 7.5694,C 0.1357,E1 7.4951,E2 332.441} C_DIS
LIN {X -63.092,Y 122.9989,Z 175,A 117.7393,B 7.5694,C 0.1323,E1 7.4997,E2 334.3317} C_DIS
LIN {X -59.2771,Y 124.882,Z 175,A 115.9785,B 7.5694,C 0.13,E1 7.5042,E2 336.0908} C_DIS
LIN {X -55.2566,Y 126.7125,Z 175,A 114.0956,B 7.5695,C 0.1286,E1 7.509,E2 337.9787} C_DIS
LIN {X -51.7467,Y 128.1853,Z 175,A 112.6139,B 7.5695,C 0.1255,E1 7.5128,E2 339.4475} C_DIS
LIN {X -48.6288,Y 129.4003,Z 175,A 110.7184,B 7.5695,C 0.1317,E1 7.5179,E2 341.4042} C_DIS
LIN {X -44.4974,Y 130.8811,Z 175,A 109.2289,B 7.5695,C 0.125,E1 7.5217,E2 342.8523} C_DIS
LIN {X -40.6689,Y 132.1185,Z 175,A 107.7036,B 7.5696,C 0.1214,E1 7.5257,E2 344.3588} C_DIS
LIN {X -36.5955,Y 133.3057,Z 175,A 105.9254,B 7.5696,C 0.1203,E1 7.5305,E2 346.1384} C_DIS
LIN {X -32.8624,Y 134.2741,Z 175,A 104.3756,B 7.5696,C 0.1184,E1 7.5347,E2 347.6811} C_DIS
LIN {X -29.2194,Y 135.1128,Z 175,A 102.8204,B 7.5696,C 0.1175,E1 7.5389,E2 349.236} C_DIS
LIN {X -24.5504,Y 136.0389,Z 175,A 101.0109,B 7.5698,C 0.1139,E1 7.5438,E2 351.0242} C_DIS
LIN {X -22.5845,Y 136.379,Z 175,A 99.517,B 7.5696,C 0.124,E1 7.5482,E2 352.5995} C_DIS
LIN {X -18.5556,Y 136.9866,Z 175,A 98.341,B 7.5697,C 0.1152,E1 7.5512,E2 353.7119} C_DIS
LIN {X -11.0222,Y 137.7976,Z 175,A 95.4894,B 7.5698,C 0.1097,E1 7.5591,E2 356.5263} C_DIS
LIN {X -4.5006,Y 138.1648,Z 175,A 92.283,B 7.5698,C 0.1173,E1 7.5682,E2 359.7931} C_DIS
LIN {X -0.8556,Y 138.2339,Z 175,A 90.5179,B 7.5696,C 0.1214,E1 7.5732,E2 361.5886} C_DIS
LIN {X 2.8925,Y 138.2075,Z 175,A 89.2186,B 7.5697,C 0.1173,E1 7.5767,E2 362.8562} C_DIS
LIN {X 8.3092,Y 137.9866,Z 175,A 87.0592,B 7.5697,C 0.1162,E1 7.5827,E2 365.0038} C_DIS
LIN {X 11.821,Y 137.7301,Z 175,A 85.0641,B 7.5696,C 0.1254,E1 7.5884,E2 367.0639} C_DIS
LIN {X 16.5291,Y 137.2446,Z 175,A 83.65,B 7.5697,C 0.117,E1 7.5922,E2 368.4103} C_DIS
LIN {X 21.4132,Y 136.568,Z 175,A 81.548,B 7.5697,C 0.1188,E1 7.598,E2 370.5188} C_DIS
LIN {X 25.5828,Y 135.8489,Z 175,A 79.5559,B 7.5697,C 0.1237,E1 7.6035,E2 372.5397} C_DIS
LIN {X 28.9494,Y 135.1711,Z 175,A 78.5298,B 7.5697,C 0.1178,E1 7.6062,E2 373.5166} C_DIS
LIN {X 31.3935,Y 134.6257,Z 175,A 77.279,B 7.5697,C 0.1221,E1 7.6097,E2 374.7934} C_DIS
LIN {X 35.5109,Y 133.5972,Z 175,A 75.7731,B 7.5697,C 0.119,E1 7.6137,E2 376.2677} C_DIS
LIN {X 38.0747,Y 132.8916,Z 175,A 74.4792,B 7.5697,C 0.1232,E1 7.6172,E2 377.5852} C_DIS
LIN {X 41.5225,Y 131.8537,Z 175,A 73.0222,B 7.5696,C 0.1238,E1 7.6211,E2 379.0374} C_DIS
LIN {X 45.1121,Y 130.668,Z 175,A 71.5804,B 7.5696,C 0.1231,E1 7.6249,E2 380.4636} C_DIS
LIN {X 48.0101,Y 129.6321,Z 175,A 70.2227,B 7.5696,C 0.1258,E1 7.6285,E2 381.8313} C_DIS
LIN {X 51.299,Y 128.3657,Z 175,A 68.6453,B 7.5696,C 0.1294,E1 7.6326,E2 383.4228} C_DIS
LIN {X 56.0546,Y 126.3615,Z 175,A 66.6785,B 7.5696,C 0.1288,E1 7.6376,E2 385.3683} C_DIS
LIN {X 59.4722,Y 124.7888,Z 175,A 65.3945,B 7.5696,C 0.1258,E1 7.6408,E2 386.6181} C_DIS
LIN {X 64.3556,Y 122.3418,Z 175,A 62.9457,B 7.5695,C 0.132,E1 7.6469,E2 389.0898} C_DIS
LIN {X 68.0304,Y 120.3399,Z 175,A 61.0822,B 7.5694,C 0.1367,E1 7.6515,E2 390.9695} C_DIS
LIN {X 71.6478,Y 118.2216,Z 175,A 59.2219,B 7.5693,C 0.1415,E1 7.656,E2 392.845} C_DIS
LIN {X 74.4767,Y 116.46,Z 175,A 57.2087,B 7.569,C 0.1549,E1 7.6609,E2 394.9358} C_DIS
LIN {X 79.9671,Y 112.7613,Z 175,A 55.2923,B 7.5692,C 0.1445,E1 7.6651,E2 396.751} C_DIS
LIN {X 83.5308,Y 110.1473,Z 175,A 53.4736,B 7.5692,C 0.1474,E1 7.6691,E2 398.5683} C_DIS
LIN {X 87.0713,Y 107.3705,Z 175,A 51.6424,B 7.5692,C 0.1501,E1 7.6731,E2 400.3957} C_DIS
LIN {X 90.5366,Y 104.4654,Z 175,A 49.9322,B 7.5692,C 0.1506,E1 7.6767,E2 402.0859} C_DIS
LIN {X 93.1555,Y 102.1366,Z 175,A 48.3841,B 7.569,C 0.1551,E1 7.68,E2 403.6462} C_DIS
LIN {X 97.6577,Y 97.8406,Z 175,A 46.1086,B 7.569,C 0.1546,E1 7.6845,E2 405.8846} C_DIS
LIN {X 102.9843,Y 92.2168,Z 175,A 42.6753,B 7.5688,C 0.1655,E1 7.6911,E2 409.3469} C_DIS
LIN {X 105.7279,Y 89.0584,Z 175,A 40.9402,B 7.5688,C 0.1693,E1 7.6942,E2 411.0828} C_DIS
LIN {X 108.3732,Y 85.82,Z 175,A 39.1072,B 7.5686,C 0.1751,E1 7.6975,E2 412.9288} C_DIS
LIN {X 111.5429,Y 81.6576,Z 175,A 37.0887,B 7.5686,C 0.1772,E1 7.7008,E2 414.9295} C_DIS
LIN {X 114.1823,Y 77.9246,Z 175,A 35.0356,B 7.5684,C 0.1847,E1 7.7041,E2 417.0032} C_DIS
LIN {X 115.9723,Y 75.234,Z 175,A 33.9286,B 7.5684,C 0.1834,E1 7.7057,E2 418.0819} C_DIS
LIN {X 121.1026,Y 66.6633,Z 175,A 29.8288,B 7.5682,C 0.1929,E1 7.7116,E2 422.1789} C_DIS
LIN {X 123.0346,Y 63.0219,Z 175,A 28.3018,B 7.5682,C 0.1937,E1 7.7135,E2 423.6841} C_DIS
LIN {X 124.3388,Y 60.4129,Z 175,A 26.9527,B 7.568,C 0.1996,E1 7.7152,E2 425.0515} C_DIS
LIN {X 126.0065,Y 56.8483,Z 175,A 25.4017,B 7.568,C 0.2022,E1 7.717,E2 426.5933} C_DIS
LIN {X 127.2079,Y 54.111,Z 175,A 24.048,B 7.5678,C 0.2077,E1 7.7185,E2 427.9622} C_DIS
LIN {X 128.7503,Y 50.3249,Z 175,A 22.6021,B 7.5678,C 0.2074,E1 7.7199,E2 429.3779} C_DIS
LIN {X 129.8435,Y 47.4363,Z 175,A 21.2551,B 7.5676,C 0.2122,E1 7.7213,E2 430.7343} C_DIS
LIN {X 131.0564,Y 43.9719,Z 175,A 19.8036,B 7.5676,C 0.2149,E1 7.7226,E2 432.1779} C_DIS
LIN {X 132.1108,Y 40.6941,Z 175,A 18.3917,B 7.5675,C 0.2185,E1 7.7238,E2 433.5889} C_DIS
LIN {X 133.0883,Y 37.3731,Z 175,A 17.0418,B 7.5675,C 0.2208,E1 7.7248,E2 434.9291} C_DIS
LIN {X 134.0001,Y 33.9589,Z 175,A 15.5962,B 7.5673,C 0.2245,E1 7.7258,E2 436.3734} C_DIS
LIN {X 134.9591,Y 29.9314,Z 175,A 13.9181,B 7.5672,C 0.2286,E1 7.7269,E2 438.048} C_DIS
LIN {X 135.8446,Y 25.6053,Z 175,A 12.0759,B 7.567,C 0.234,E1 7.7279,E2 439.8931} C_DIS
LIN {X 136.5623,Y 21.4498,Z 175,A 10.4377,B 7.567,C 0.2367,E1 7.7286,E2 441.5187} C_DIS
LIN {X 137.0113,Y 18.3668,Z 175,A 8.3161,B 7.5663,C 0.2568,E1 7.7295,E2 443.7458} C_DIS
LIN {X 137.6941,Y 12.248,Z 175,A 6.5063,B 7.5665,C 0.2495,E1 7.7299,E2 445.4645} C_DIS
LIN {X 137.9586,Y 8.7642,Z 175,A 4.6536,B 7.5661,C 0.2616,E1 7.7303,E2 447.3694} C_DIS
LIN {X 138.1759,Y 4.0983,Z 175,A 3.3573,B 7.5663,C 0.2546,E1 7.7303,E2 448.5867} C_DIS
LIN {X 138.2365,Y 0.5259,Z 175,A 1.8234,B 7.5662,C 0.2599,E1 7.7304,E2 450.1286} C_DIS
LIN {X 138.192,Y -3.5199,Z 175,A 0.16,B 7.566,C 0.2645,E1 7.7304,E2 451.7917} C_DIS
LIN {X 137.8976,Y -9.6797,Z 175,A -2.8801,B 7.5654,C 0.2814,E1 7.7298,E2 454.8952} C_DIS
LIN {X 137.4765,Y -14.4776,Z 175,A -4.4048,B 7.5655,C 0.2778,E1 7.7294,E2 456.3622} C_DIS
LIN {X 136.952,Y -18.8134,Z 175,A -6.4223,B 7.5652,C 0.2871,E1 7.7287,E2 458.4077} C_DIS
LIN {X 136.4061,Y -22.4217,Z 175,A -7.6643,B 7.5652,C 0.2861,E1 7.7281,E2 459.6167} C_DIS
LIN {X 135.3043,Y -28.3303,Z 175,A -9.9873,B 7.5651,C 0.2898,E1 7.7269,E2 461.9208} C_DIS
LIN {X 134.4113,Y -32.2933,Z 175,A -11.3963,B 7.5651,C 0.2891,E1 7.726,E2 463.2962} C_DIS
LIN {X 133.6202,Y -35.4247,Z 175,A -12.9305,B 7.5648,C 0.2968,E1 7.725,E2 464.8567} C_DIS
LIN {X 131.8491,Y -41.5371,Z 175,A -15.6195,B 7.5645,C 0.3051,E1 7.7228,E2 467.5548} C_DIS
LIN {X 130.7577,Y -44.8534,Z 175,A -16.8347,B 7.5645,C 0.3045,E1 7.7218,E2 468.7418} C_DIS
LIN {X 129.7918,Y -47.5797,Z 175,A -18.1087,B 7.5643,C 0.3093,E1 7.7205,E2 470.0266} C_DIS
LIN {X 127.9939,Y -52.2215,Z 175,A -20.215,B 7.5641,C 0.3158,E1 7.7184,E2 472.1404} C_DIS
LIN {X 126.7221,Y -55.2344,Z 175,A -22.3895,B 7.5632,C 0.3354,E1 7.7158,E2 474.4203} C_DIS
LIN {X 123.9141,Y -61.2738,Z 175,A -24.1675,B 7.5637,C 0.3235,E1 7.7138,E2 476.0761} C_DIS
LIN {X 122.1894,Y -64.6458,Z 175,A -25.7928,B 7.5635,C 0.3287,E1 7.7117,E2 477.7101} C_DIS
LIN {X 119.9947,Y -68.6368,Z 175,A -27.6687,B 7.5633,C 0.3333,E1 7.7091,E2 479.5864} C_DIS
LIN {X 117.6184,Y -72.6346,Z 175,A -29.6363,B 7.5631,C 0.3389,E1 7.7063,E2 481.5611} C_DIS
LIN {X 115.1783,Y -76.4449,Z 175,A -31.4688,B 7.5629,C 0.3427,E1 7.7035,E2 483.3899} C_DIS
LIN {X 112.6756,Y -80.088,Z 175,A -33.279,B 7.5627,C 0.3467,E1 7.7006,E2 485.1991} C_DIS
Enddeposition()
END
